// TIA Portal V16 program export: 3 tag tables, 3 data types, 3 data blocks, 6 code blocks (in call order from the OBs), 9 instance data blocks

VAR_GLOBAL   // PLC tag table "Entradas PLC"
   "Rele Emergencia" AT %I0.0 : Bool;
   "Rele Barrera" AT %I0.1 : Bool;
   "Pulsador Rearme" AT %I0.2 : Bool;
   "Marcha 1" AT %I0.3 : Bool;
   "Marcha 2" AT %I0.4 : Bool;
   "Marcha 3" AT %I0.5 : Bool;
   Caudalímetro AT %I0.6 : Bool;
   Presostato AT %I0.7 : Bool;
   "Final Soldadura" AT %I1.1 : Bool;
   "Soldadura RDY" AT %I1.0 : Bool;
   "Acuse error soldadura" AT %I1.2 : Bool;
   "Fibra óptica Tornillo 1" AT %I1.3 : Bool;
   "Fibra óptica Tornillo 2" AT %I1.4 : Bool;
   "Cajón rechazo" AT %I1.5 : Bool;
   "Pinza 1 RE" AT %I2.0 : Bool;
   "Pinza 1 AV" AT %I2.1 : Bool;
   "Pinza 2 RE" AT %I2.2 : Bool;
   "Pinza 2 AV" AT %I2.3 : Bool;
   "Pinza 3 RE" AT %I2.4 : Bool;
   "Pinza 3 AV" AT %I2.5 : Bool;
   "Libre I 2.6" AT %I2.6 : Bool;
   "Libre I 2.7" AT %I2.7 : Bool;
   "Selector acuse pieza mala" AT %I3.0 : Bool;
   RobotOK AT %I3.1 : Bool;
   RobotNOK AT %I3.2 : Bool;
   RobotAuto AT %I3.3 : Bool;
   "Libre I 3.4" AT %I3.4 : Bool;
   "Libre I 3.5" AT %I3.5 : Bool;
   "Libre I 3.6" AT %I3.6 : Bool;
   "Libre I 3.7" AT %I3.7 : Bool;
   Tag_71 AT %IW64 : Word;
END_VAR

VAR_GLOBAL   // PLC tag table "Salidas PLC"
   Rearme AT %Q0.0 : Bool;
   "Marcha Soldadura" AT %Q0.1 : Bool;
   "Programa 1" AT %Q0.2 : Bool;
   "Programa 2" AT %Q0.3 : Bool;
   "Programa 4" AT %Q0.4 : Bool;
   "Programa 8" AT %Q0.5 : Bool;
   "Programa 16" AT %Q0.6 : Bool;
   "Reset error" AT %Q0.7 : Bool;
   Fluorescent AT %Q1.0 : Bool;
   "Piloto 1 Rojo" AT %Q2.0 : Bool;
   "Piloto 1 Ambar" AT %Q2.1 : Bool;
   "Piloto 1 Verde" AT %Q2.2 : Bool;
   "Piloto 2 Rojo" AT %Q2.3 : Bool;
   "Piloto 2 Ambar" AT %Q2.4 : Bool;
   "Piloto 2 Verde" AT %Q2.5 : Bool;
   "Piloto 3 Rojo" AT %Q2.6 : Bool;
   "Piloto 3 Ambar" AT %Q2.7 : Bool;
   "Piloto 3 Verde" AT %Q3.0 : Bool;
   "Baliza Roja" AT %Q3.1 : Bool;
   "Baliza Ambar" AT %Q3.2 : Bool;
   "Baliza Verde" AT %Q3.3 : Bool;
   "Pinza 1" AT %Q4.0 : Bool;
   "Pinza 2" AT %Q4.1 : Bool;
   "Pinza 3" AT %Q4.2 : Bool;
   "Piloto Marcha 1" AT %Q3.5 : Bool;
   "Piloto Marcha 2" AT %Q3.6 : Bool;
   "Piloto Marcha 3" AT %Q3.7 : Bool;
   "Piloto rearme" AT %Q3.4 : Bool;
   "Libre Q 4.7" AT %Q4.7 : Bool;
   Tag_46 AT %Q1.1 : Bool;
   bNotReady AT %Q4.4 : Bool;
   bRobotReset AT %Q4.5 : Bool;
END_VAR

VAR_GLOBAL   // PLC tag table "Tabla de variables estándar"
   System_Byte AT %MB1001 : Byte;
   FirstScan AT %M1001.0 : Bool;
   DiagStatusUpdate AT %M1001.1 : Bool;
   AlwaysTRUE AT %M1001.2 : Bool;
   AlwaysFALSE AT %M1001.3 : Bool;
   Clock_Byte AT %MB1000 : Byte;
   Clock_10Hz AT %M1000.0 : Bool;
   Clock_5Hz AT %M1000.1 : Bool;
   "Clock_2.5Hz" AT %M1000.2 : Bool;
   Clock_2Hz AT %M1000.3 : Bool;
   "Clock_1.25Hz" AT %M1000.4 : Bool;
   Clock_1Hz AT %M1000.5 : Bool;
   "Clock_0.625Hz" AT %M1000.6 : Bool;
   "Clock_0.5Hz" AT %M1000.7 : Bool;
   Tag_1 AT %MW100 : Word;
   Tag_2 AT %M10.0 : Bool;
   bStartShortBolt AT %M20.0 : Bool;
   bStartMediumBolt AT %M20.1 : Bool;
   bStartLongBolt AT %M20.2 : Bool;
   bStartWeldingGripper_3 AT %M20.3 : Bool;
   bRetractGripper_3 AT %M20.4 : Bool;
   Tag_8 AT %M20.5 : Bool;
   Tag_9 AT %M20.6 : Bool;
   Tag_10 AT %M20.7 : Bool;
   bGripper_3_Conditions AT %M29.0 : Bool;
   bStartSmallNut AT %M21.0 : Bool;
   bStartBigNut AT %M21.1 : Bool;
   bStartWeldingGripper_2 AT %M21.2 : Bool;
   bRetractGripper_2 AT %M21.3 : Bool;
   Tag_16 AT %M21.4 : Bool;
   Tag_17 AT %M21.5 : Bool;
   Tag_18 AT %M21.6 : Bool;
   Tag_19 AT %M21.7 : Bool;
   bGripper_2_Conditions AT %M29.1 : Bool;
   bStartSpot AT %M22.0 : Bool;
   bStartWeldingGripper_1 AT %M22.1 : Bool;
   bRetractGripper_1 AT %M22.2 : Bool;
   Tag_24 AT %M22.3 : Bool;
   Tag_25 AT %M22.4 : Bool;
   Tag_26 AT %M22.5 : Bool;
   Tag_27 AT %M22.6 : Bool;
   Tag_28 AT %M22.7 : Bool;
   bGripper_1_Conditions AT %M29.2 : Bool;
   bCycleConditions AT %M29.3 : Bool;
   bEndOfCycle AT %M23.0 : Bool;
   bWeldingNOK AT %M23.1 : Bool;
   bToScrap AT %M23.2 : Bool;
   bScraped AT %M23.3 : Bool;
   bScrapBoxFull AT %M23.4 : Bool;
   bConsecutiveNOKtoBlock AT %M23.5 : Bool;
   bRobotAuto AT %M23.6 : Bool;
   bProductionCompleted AT %M23.7 : Bool;
   bAction_1 AT %M24.0 : Bool;
   bAction_2 AT %M24.1 : Bool;
   bAction_3 AT %M24.2 : Bool;
   bAction_4 AT %M24.3 : Bool;
   bAction_5 AT %M24.4 : Bool;
   bAction_6 AT %M24.5 : Bool;
   bEndSequence AT %M24.6 : Bool;
   BWelderProgNumber AT %MB12 : Byte;
   bWelderProg_Bit_0 AT %M12.0 : Bool;
   bWelderProg_Bit_1 AT %M12.1 : Bool;
   bWelderProg_Bit_2 AT %M12.2 : Bool;
   bWelderProg_Bit_3 AT %M12.3 : Bool;
   bWelderProg_Bit_4 AT %M12.4 : Bool;
   Tag_53 AT %MW20 : Int;
   Tag_54 AT %MW22 : Int;
   Tag_55 AT %MW24 : Int;
   "Alarmes 1" AT %MW200 : Word;
   "Alarmes 2" AT %MW202 : Word;
   bAnyAlarm AT %M210.0 : Bool;
   Tag_59 AT %MD200 : DWord;
   bEmergenciesNOK AT %M200.0 : Bool;
   bPressureFault AT %M200.1 : Bool;
   bFlowFault AT %M200.2 : Bool;
   "Alarma barrera cajon rechazo" AT %M200.3 : Bool;
   "Alarma pinza 1 no avanza" AT %M201.0 : Bool;
   "Alarma pinza 1 No retrocede" AT %M201.1 : Bool;
   "Alarma pinza 2 No avanza" AT %M201.2 : Bool;
   "Alarma pinza 2 No retrocede" AT %M201.3 : Bool;
   "Alarma pinza3 no avanza" AT %M201.4 : Bool;
   "Alarma pinza 3 No retrocede" AT %M201.5 : Bool;
   bWelderNotReady AT %M200.4 : Bool;
   bWelderNotResponding AT %M200.5 : Bool;
   "Alarma barrera obstruida" AT %M202.0 : Bool;
   Tag_73 AT %M200.6 : Bool;
   "Aviso perno corto incorreto" AT %M202.1 : Bool;
   "Aviso perno medio incorrecto" AT %M202.2 : Bool;
   "Aviso perno largo incorrecto" AT %M202.3 : Bool;
   "Aviso pieza mala" AT %M202.4 : Bool;
   "Aviso tirar pieza mala" AT %M202.5 : Bool;
   Tag_79 AT %M202.6 : Bool;
   bInitConditions AT %M29.4 : Bool;
   "Alarmes 6" AT %MW210 : Word;
   Tag_56 AT %M200.7 : Bool;
   Tag_57 AT %M5.0 : Bool;
   Tag_60 AT %M5.1 : Bool;
   Tag_61 AT %M5.2 : Bool;
   Tag_62 AT %M5.3 : Bool;
   Tag_63 AT %M5.4 : Bool;
   Tag_64 AT %M5.5 : Bool;
   Tag_58 AT %M7.0 : Bool;
   Tag_65 AT %M6.5 : Bool;
   Tag_66 AT %M6.4 : Bool;
   Tag_67 AT %M6.2 : Bool;
   Tag_68 AT %M6.3 : Bool;
   Tag_69 AT %M6.0 : Bool;
   Tag_70 AT %M6.1 : Bool;
   bTemp_PAP AT %M100.0 : Bool;
   bRedLamp_3_NonInverted AT %M50.0 : Bool;
   bRedLamp_1_Inverted AT %M50.1 : Bool;
   bAmberLamp_3_NonInverted AT %M50.2 : Bool;
   bGreenLamp_3_NonInverted AT %M50.4 : Bool;
   bAmberLamp_1_Inverted AT %M50.3 : Bool;
   bGreenLamp_1_Inverted AT %M50.5 : Bool;
   bRedLamp_1_NonInverted AT %M50.6 : Bool;
   bRedLamp_3_Inverted AT %M50.7 : Bool;
   bAmberLamp_1_NonInverted AT %M51.0 : Bool;
   bAmberLamp_3_Inverted AT %M51.1 : Bool;
   bGreenLamp_1_NonInverted AT %M51.2 : Bool;
   bGreenLamp_3_Inverted AT %M51.3 : Bool;
   bStartLamp_1_NonInverted AT %M51.4 : Bool;
   bStartLamp_3_NonInverted AT %M51.5 : Bool;
   bStartLamp_3_Inverted AT %M51.6 : Bool;
   bStartLamp_1_Inverted AT %M51.7 : Bool;
   bGripper_3_NonInverted AT %M52.0 : Bool;
   bGripper_1_NonInverted AT %M52.1 : Bool;
   bGripper_3_Inverted AT %M52.3 : Bool;
   bGripper_1_Inverted AT %M52.2 : Bool;
END_VAR

TYPE "udtCounters"
// stored: IsFailsafeCompliant false
   STRUCT
      diPreselectionValue : DInt;
      diTotalOK : DInt;
      diPartialOK : DInt;
      diConsecutiveOK : DInt;
      diTotalNOK : DInt;
      diPartialNOK : DInt;
      diConsecutiveNOK : DInt;
      diScrapBox : DInt;
      stSettings : Struct
         diScrapBoxSize : DInt;
         diNOKValueToBlock : DInt;
         diOKValueToResetNOK : DInt;
      END_STRUCT;
      stButtons : Struct
         bResetTotalOK : Bool;
         bResetPartialOK : Bool;
         bResetConsecutiveOK : Bool;
         bResetTotalNOK : Bool;
         bResetPartialNOK : Bool;
         bResetConsecutiveNOK : Bool;
         bResetScrapBox : Bool;
      END_STRUCT;
   END_STRUCT;
END_TYPE

TYPE "udtProgram"
// stored: IsFailsafeCompliant false
   STRUCT
      strName : String[12];
      udtStep { S7_SetPoint := 'True'} : Array[1..10] of "udtStep";
      udtCounter { S7_SetPoint := 'True'} : "udtCounters";
   END_STRUCT;
END_TYPE

TYPE "udtStep"
// stored: IsFailsafeCompliant false
   STRUCT
      iAction : Int;
      iPG : Int;
      iLamp : Int;
   END_STRUCT;
END_TYPE

DATA_BLOCK "db_HMI"   // DB100
{ S7_Optimized_Access := 'FALSE' }
VERSION : 0.1
// stored: AutoNumber false, IsOnlyStoredInLoadMemory false, IsWriteProtectedInAS false
   VAR
      ariScreen : Array[0..3] of Int;
      iScreenNumbver : Int;
      bLights : Bool;
      bResetCycleKey : Bool;
      diPartsCounter : DInt;
      iPart_1 : Int;
      iPart_2 : Int;
      iPart_3 : Int;
      iPart_4 : Int;
      iPart_5 : Int;
      iPart_6 : Int;
      iPart_7 : Int;
      iPart_8 : Int;
      iPart_9 : Int;
      iPart_10 : Int;
   END_VAR
BEGIN
END_DATA_BLOCK

DATA_BLOCK "db_Programs"   // DB101
{ S7_Optimized_Access := 'TRUE' }
VERSION : 0.1
// stored: AutoNumber false, IsOnlyStoredInLoadMemory false, IsRetainMemResEnabled false, IsWriteProtectedInAS false, MemoryReserve 100
   VAR RETAIN
      diProgramSelection : DInt := 8;
   END_VAR
   VAR
      bSaveKey : Bool := FALSE;
      diStepCounter : DInt := 1;
      strShortBolt : String[16] := '';
      strMediumBolt : String[16] := '';
      strLongBolt : String[16] := '';
      strSmallNut : String[16] := '';
      strBigNut : String[16] := '';
   END_VAR
   VAR RETAIN
      udtProgram { S7_SetPoint := 'True'} : Array[1..10] of "udtProgram";
      udtWorkProgram { S7_SetPoint := 'True'} : "udtProgram";
   END_VAR
   VAR
      udtWorkStep { S7_SetPoint := 'True'} : "udtStep";
   END_VAR
BEGIN
   udtProgram[1].strName := 'TCS327=178';
   udtProgram[2].strName := 'TCS327=193';
   udtProgram[3].strName := 'TCS327=192';
   udtProgram[4].strName := 'TCS327=181';
   udtProgram[5].strName := 'TCS327=186';
   udtProgram[6].strName := 'TCS327=200';
   udtProgram[7].strName := 'TCS327=188';
   udtProgram[8].strName := 'TCS327=190';
   udtProgram[9].strName := 'TCS327=197';
   udtProgram[10].strName := '191.33476980';
   udtProgram[1].udtStep[1..4].iAction := 2;
   udtProgram[1].udtStep[5..7].iAction := 1;
   udtProgram[1].udtStep[8..10].iAction := 0;
   udtProgram[2].udtStep[1].iAction := 6;
   udtProgram[2].udtStep[2].iAction := 5;
   udtProgram[2].udtStep[3..4].iAction := 3;
   udtProgram[2].udtStep[5..10].iAction := 0;
   udtProgram[3].udtStep[1..2].iAction := 1;
   udtProgram[3].udtStep[3..10].iAction := 0;
   udtProgram[4].udtStep[1..3].iAction := 6;
   udtProgram[4].udtStep[4].iAction := 1;
   udtProgram[4].udtStep[5..10].iAction := 0;
   udtProgram[5].udtStep[1..2].iAction := 2;
   udtProgram[5].udtStep[3..10].iAction := 0;
   udtProgram[6].udtStep[1].iAction := 5;
   udtProgram[6].udtStep[2].iAction := 1;
   udtProgram[6].udtStep[3..10].iAction := 0;
   udtProgram[7].udtStep[1].iAction := 5;
   udtProgram[7].udtStep[2].iAction := 1;
   udtProgram[7].udtStep[3..10].iAction := 0;
   udtProgram[8].udtStep[1].iAction := 6;
   udtProgram[8].udtStep[2].iAction := 4;
   udtProgram[8].udtStep[3..7].iAction := 1;
   udtProgram[8].udtStep[8..10].iAction := 0;
   udtProgram[9].udtStep[1..3].iAction := 4;
   udtProgram[9].udtStep[4..10].iAction := 0;
   udtProgram[10].udtStep[1..10].iAction := 0;
   udtProgram[1].udtStep[1..7].iPG := 3;
   udtProgram[1].udtStep[8..10].iPG := 0;
   udtProgram[2].udtStep[1].iPG := 22;
   udtProgram[2].udtStep[2].iPG := 23;
   udtProgram[2].udtStep[3..4].iPG := 3;
   udtProgram[2].udtStep[5].iPG := 9;
   udtProgram[2].udtStep[6..7].iPG := 1;
   udtProgram[2].udtStep[8..10].iPG := 0;
   udtProgram[3].udtStep[1..2].iPG := 3;
   udtProgram[3].udtStep[3..10].iPG := 0;
   udtProgram[4].udtStep[1..3].iPG := 22;
   udtProgram[4].udtStep[4].iPG := 3;
   udtProgram[4].udtStep[5..10].iPG := 0;
   udtProgram[5].udtStep[1..3].iPG := 3;
   udtProgram[5].udtStep[4..10].iPG := 0;
   udtProgram[6].udtStep[1].iPG := 5;
   udtProgram[6].udtStep[2].iPG := 3;
   udtProgram[6].udtStep[3..10].iPG := 0;
   udtProgram[7].udtStep[1].iPG := 5;
   udtProgram[7].udtStep[2].iPG := 3;
   udtProgram[7].udtStep[3..10].iPG := 0;
   udtProgram[8].udtStep[1].iPG := 1;
   udtProgram[8].udtStep[2].iPG := 2;
   udtProgram[8].udtStep[3..7].iPG := 3;
   udtProgram[8].udtStep[8..10].iPG := 0;
   udtProgram[9].udtStep[1..3].iPG := 1;
   udtProgram[9].udtStep[4..10].iPG := 0;
   udtProgram[10].udtStep[1..10].iPG := 0;
   udtProgram[1].udtStep[1].iLamp := 2;
   udtProgram[1].udtStep[2].iLamp := 1;
   udtProgram[1].udtStep[3].iLamp := 3;
   udtProgram[1].udtStep[4].iLamp := 4;
   udtProgram[1].udtStep[5].iLamp := 5;
   udtProgram[1].udtStep[6].iLamp := 6;
   udtProgram[1].udtStep[7].iLamp := 7;
   udtProgram[1].udtStep[8..10].iLamp := 0;
   udtProgram[2].udtStep[1..2].iLamp := 2;
   udtProgram[2].udtStep[3].iLamp := 3;
   udtProgram[2].udtStep[4].iLamp := 4;
   udtProgram[2].udtStep[5].iLamp := 5;
   udtProgram[2].udtStep[6].iLamp := 6;
   udtProgram[2].udtStep[7].iLamp := 7;
   udtProgram[2].udtStep[8..10].iLamp := 0;
   udtProgram[3].udtStep[1].iLamp := 1;
   udtProgram[3].udtStep[2].iLamp := 2;
   udtProgram[3].udtStep[3..10].iLamp := 0;
   udtProgram[4].udtStep[1].iLamp := 1;
   udtProgram[4].udtStep[2].iLamp := 2;
   udtProgram[4].udtStep[3].iLamp := 3;
   udtProgram[4].udtStep[4..10].iLamp := 0;
   udtProgram[5].udtStep[1].iLamp := 1;
   udtProgram[5].udtStep[2].iLamp := 2;
   udtProgram[5].udtStep[3].iLamp := 3;
   udtProgram[5].udtStep[4..10].iLamp := 0;
   udtProgram[6].udtStep[1].iLamp := 1;
   udtProgram[6].udtStep[2].iLamp := 2;
   udtProgram[6].udtStep[3..10].iLamp := 0;
   udtProgram[7].udtStep[1].iLamp := 1;
   udtProgram[7].udtStep[2].iLamp := 2;
   udtProgram[7].udtStep[3..10].iLamp := 0;
   udtProgram[8].udtStep[1].iLamp := 7;
   udtProgram[8].udtStep[2].iLamp := 1;
   udtProgram[8].udtStep[3].iLamp := 6;
   udtProgram[8].udtStep[4].iLamp := 5;
   udtProgram[8].udtStep[5].iLamp := 3;
   udtProgram[8].udtStep[6].iLamp := 2;
   udtProgram[8].udtStep[7].iLamp := 4;
   udtProgram[8].udtStep[8..10].iLamp := 0;
   udtProgram[9].udtStep[1].iLamp := 1;
   udtProgram[9].udtStep[2].iLamp := 2;
   udtProgram[9].udtStep[3].iLamp := 3;
   udtProgram[9].udtStep[4..10].iLamp := 0;
   udtProgram[10].udtStep[1..10].iLamp := 0;
   udtWorkProgram.strName := 'TCS327=190';
   udtWorkProgram.udtStep[1].iAction := 6;
   udtWorkProgram.udtStep[2].iAction := 4;
   udtWorkProgram.udtStep[3..7].iAction := 1;
   udtWorkProgram.udtStep[8..10].iAction := 0;
   udtWorkProgram.udtStep[1].iPG := 1;
   udtWorkProgram.udtStep[2].iPG := 2;
   udtWorkProgram.udtStep[3..7].iPG := 3;
   udtWorkProgram.udtStep[8..10].iPG := 0;
   udtWorkProgram.udtStep[1].iLamp := 7;
   udtWorkProgram.udtStep[2].iLamp := 1;
   udtWorkProgram.udtStep[3].iLamp := 6;
   udtWorkProgram.udtStep[4].iLamp := 5;
   udtWorkProgram.udtStep[5].iLamp := 3;
   udtWorkProgram.udtStep[6].iLamp := 2;
   udtWorkProgram.udtStep[7].iLamp := 4;
   udtWorkProgram.udtStep[8..10].iLamp := 0;
   udtWorkStep.iAction := 6;
   udtWorkStep.iPG := 1;
   udtWorkStep.iLamp := 7;
END_DATA_BLOCK

DATA_BLOCK "db_Settings"   // DB2
{ S7_Optimized_Access := 'TRUE' }
VERSION : 0.1
// stored: AutoNumber true, IsOnlyStoredInLoadMemory false, IsRetainMemResEnabled false, IsWriteProtectedInAS false, MemoryReserve 100
   VAR RETAIN
      bIsInverted : Bool;
   END_VAR
   VAR
      bBypasRobot : Bool;
   END_VAR
   VAR RETAIN
      iSerialNumber : Int;
   END_VAR
BEGIN
END_DATA_BLOCK

ORGANIZATION_BLOCK "Main"   // OB1, LAD, ProgramCycle
TITLE = "Main Program Sweep (Cycle)"
{ S7_Optimized_Access := 'TRUE' }
VERSION : 0.1
// stored: AutoNumber true, IsIECCheckEnabled false, SetENOAutomatically false
   VAR_INPUT
      Initial_Call : Bool;   // Initial call of this OB
      Remanence : Bool;   // =True, if remanent data are available
   END_VAR
BEGIN

REGION Network 1
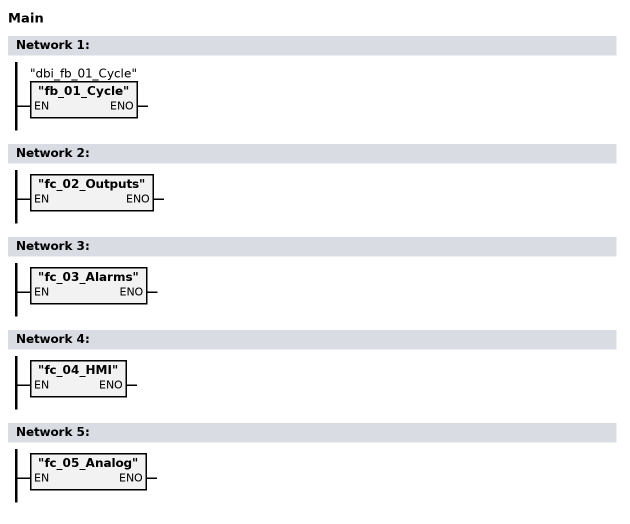
   RUNG wire#powerrail
      "dbi_fb_01_Cycle"()
   END_RUNG
   // the same network as SCL:
   "dbi_fb_01_Cycle"();   // "fb_01_Cycle"
END_REGION

REGION Network 2
   RUNG wire#powerrail
      "fc_02_Outputs"()
   END_RUNG
   // the same network as SCL:
   "fc_02_Outputs"();
END_REGION

REGION Network 3
   RUNG wire#powerrail
      "fc_03_Alarms"()
   END_RUNG
   // the same network as SCL:
   "fc_03_Alarms"();
END_REGION

REGION Network 4
   RUNG wire#powerrail
      "fc_04_HMI"()
   END_RUNG
   // the same network as SCL:
   "fc_04_HMI"();
END_REGION

REGION Network 5
   RUNG wire#powerrail
      "fc_05_Analog"()
   END_RUNG
   // the same network as SCL:
   "fc_05_Analog"();
END_REGION
END_ORGANIZATION_BLOCK

FUNCTION_BLOCK "fb_01_Cycle"   // FB1, LAD
{ S7_Optimized_Access := 'TRUE' }
VERSION : 0.1
// stored: AutoNumber false, IsIECCheckEnabled false, IsRetainMemResEnabled false, MemoryReserve 100, SetENOAutomatically false, UDAEnableTagReadback false
   VAR
      TON_Delay : Array[1..10] of TON_TIME;
      TP_Reset { S7_SetPoint := 'True'} : TP_TIME;
   END_VAR
   VAR_TEMP
      bBypassRobot : Bool;
      bRobotReset : Bool;
      bIsInverted : Bool;
   END_VAR
   VAR_TEMP   // added for the SCL form of the ladder/FBD networks
      _w1 : Bool;
      _w2 : Bool;
   END_VAR
BEGIN

REGION Network 1: Reseteo Ciclos por Emergencias
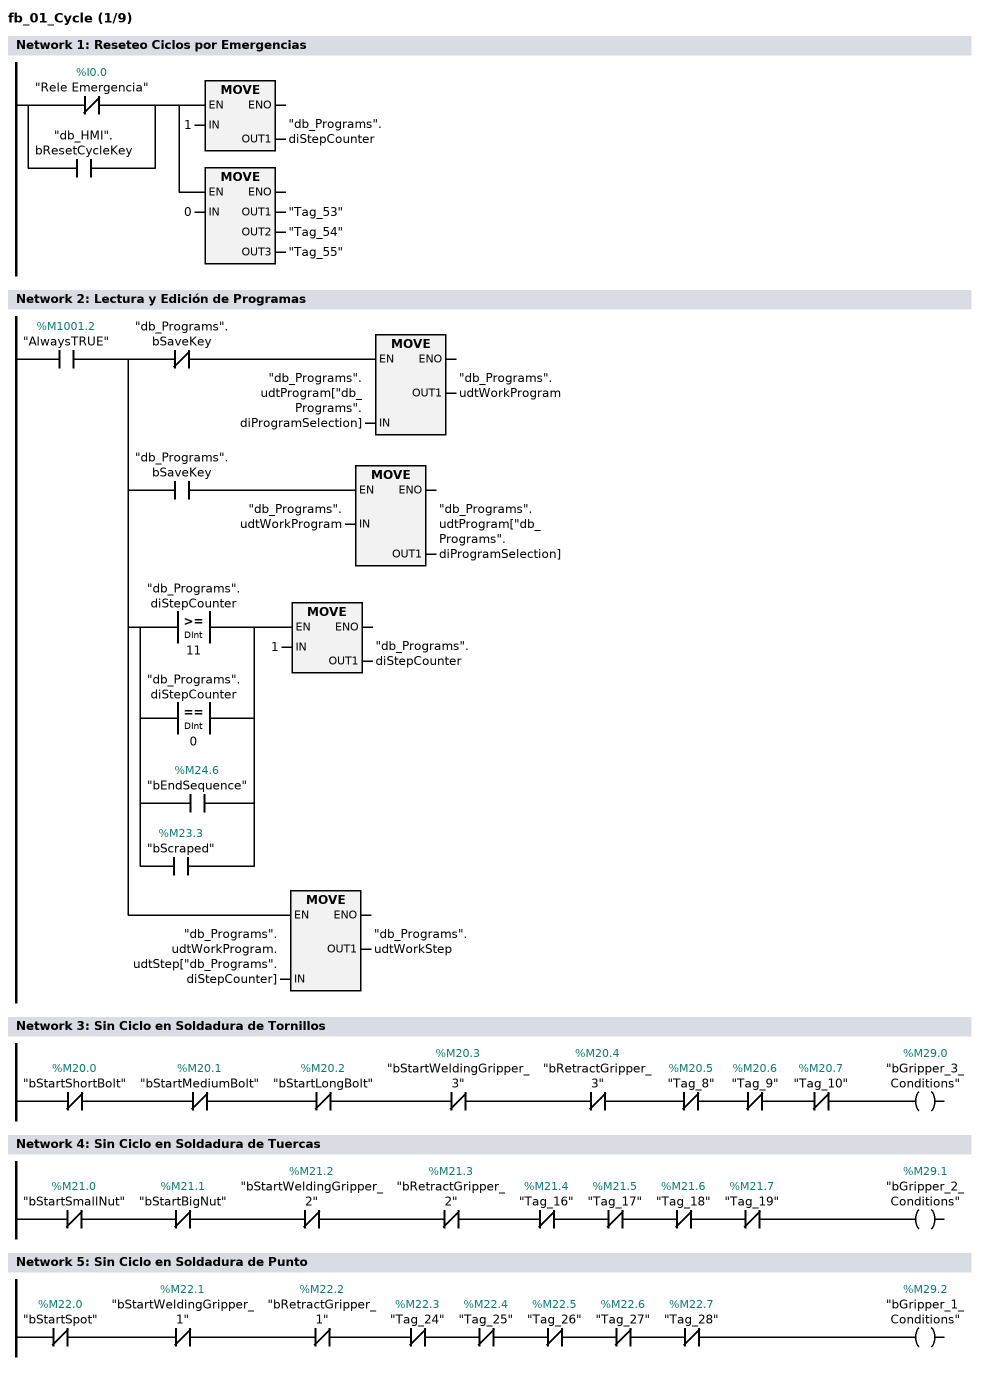
   RUNG wire#powerrail
      I_Contact( "Rele Emergencia" )
      wire#w1
      Move(in := 1, out1 => "db_Programs".diStepCounter)
   END_RUNG
   RUNG wire#powerrail
      Contact( "db_HMI".bResetCycleKey )
   END_RUNG wire#w1
   RUNG wire#w1
      Move(in := 0, out1 => "Tag_53", out2 => "Tag_54", out3 => "Tag_55")
   END_RUNG
   // the same network as SCL:
   IF NOT "Rele Emergencia" OR "db_HMI".bResetCycleKey THEN
       "db_Programs".diStepCounter := 1;
       "Tag_53" := 0;
       "Tag_54" := 0;
       "Tag_55" := 0;
   END_IF;
END_REGION

REGION Network 2: Lectura y Edición de Programas
   RUNG wire#powerrail
      Contact( "AlwaysTRUE" )
      wire#w1
      I_Contact( "db_Programs".bSaveKey )
      Move(in := "db_Programs".udtProgram["db_Programs".diProgramSelection], out1 => "db_Programs".udtWorkProgram)
   END_RUNG
   RUNG wire#w1
      Contact( "db_Programs".bSaveKey )
      Move(in := "db_Programs".udtWorkProgram, out1 => "db_Programs".udtProgram["db_Programs".diProgramSelection])
   END_RUNG
   RUNG wire#w1
      { S7_Templates := "SrcType := DInt" } GE_Contact(in1 := "db_Programs".diStepCounter, in2 := 11)
      wire#w2
      Move(in := 1, out1 => "db_Programs".diStepCounter)
   END_RUNG
   RUNG wire#w1
      { S7_Templates := "SrcType := DInt" } EQ_Contact(in1 := "db_Programs".diStepCounter, in2 := 0)
   END_RUNG wire#w2
   RUNG wire#w1
      Contact( "bEndSequence" )
   END_RUNG wire#w2
   RUNG wire#w1
      Contact( "bScraped" )
   END_RUNG wire#w2
   RUNG wire#w1
      Move(in := "db_Programs".udtWorkProgram.udtStep["db_Programs".diStepCounter], out1 => "db_Programs".udtWorkStep)
   END_RUNG
   // the same network as SCL:
   IF "AlwaysTRUE" AND NOT "db_Programs".bSaveKey THEN
       "db_Programs".udtWorkProgram := "db_Programs".udtProgram["db_Programs".diProgramSelection];
   END_IF;
   IF "AlwaysTRUE" AND "db_Programs".bSaveKey THEN
       "db_Programs".udtProgram["db_Programs".diProgramSelection] := "db_Programs".udtWorkProgram;
   END_IF;
   IF "AlwaysTRUE" AND (("db_Programs".diStepCounter >= 11) OR ("db_Programs".diStepCounter = 0) OR "bEndSequence" OR "bScraped") THEN
       "db_Programs".diStepCounter := 1;
   END_IF;
   IF "AlwaysTRUE" THEN
       "db_Programs".udtWorkStep := "db_Programs".udtWorkProgram.udtStep["db_Programs".diStepCounter];
   END_IF;
END_REGION

REGION Network 3: Sin Ciclo en Soldadura de Tornillos
   RUNG wire#powerrail
      I_Contact( "bStartShortBolt" )
      I_Contact( "bStartMediumBolt" )
      I_Contact( "bStartLongBolt" )
      I_Contact( "bStartWeldingGripper_3" )
      I_Contact( "bRetractGripper_3" )
      I_Contact( "Tag_8" )
      I_Contact( "Tag_9" )
      I_Contact( "Tag_10" )
      Coil( "bGripper_3_Conditions" )
   END_RUNG
   // the same network as SCL:
   "bGripper_3_Conditions" := NOT "bStartShortBolt" AND NOT "bStartMediumBolt" AND NOT "bStartLongBolt" AND NOT "bStartWeldingGripper_3" AND NOT "bRetractGripper_3" AND NOT "Tag_8" AND NOT "Tag_9" AND NOT "Tag_10";
END_REGION

REGION Network 4: Sin Ciclo en Soldadura de Tuercas
   RUNG wire#powerrail
      I_Contact( "bStartSmallNut" )
      I_Contact( "bStartBigNut" )
      I_Contact( "bStartWeldingGripper_2" )
      I_Contact( "bRetractGripper_2" )
      I_Contact( "Tag_16" )
      I_Contact( "Tag_17" )
      I_Contact( "Tag_18" )
      I_Contact( "Tag_19" )
      Coil( "bGripper_2_Conditions" )
   END_RUNG
   // the same network as SCL:
   "bGripper_2_Conditions" := NOT "bStartSmallNut" AND NOT "bStartBigNut" AND NOT "bStartWeldingGripper_2" AND NOT "bRetractGripper_2" AND NOT "Tag_16" AND NOT "Tag_17" AND NOT "Tag_18" AND NOT "Tag_19";
END_REGION

REGION Network 5: Sin Ciclo en Soldadura de Punto
   RUNG wire#powerrail
      I_Contact( "bStartSpot" )
      I_Contact( "bStartWeldingGripper_1" )
      I_Contact( "bRetractGripper_1" )
      I_Contact( "Tag_24" )
      I_Contact( "Tag_25" )
      I_Contact( "Tag_26" )
      I_Contact( "Tag_27" )
      I_Contact( "Tag_28" )
      Coil( "bGripper_1_Conditions" )
   END_RUNG
   // the same network as SCL:
   "bGripper_1_Conditions" := NOT "bStartSpot" AND NOT "bStartWeldingGripper_1" AND NOT "bRetractGripper_1" AND NOT "Tag_24" AND NOT "Tag_25" AND NOT "Tag_26" AND NOT "Tag_27" AND NOT "Tag_28";
END_REGION

REGION Network 6: Condiciones Ciclo Auxiliares
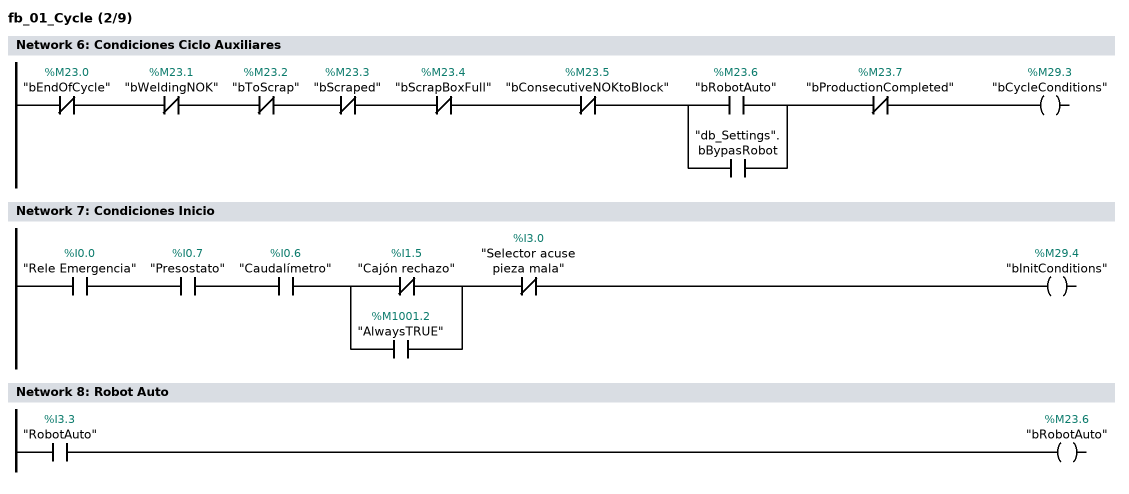
   RUNG wire#powerrail
      I_Contact( "bEndOfCycle" )
      I_Contact( "bWeldingNOK" )
      I_Contact( "bToScrap" )
      I_Contact( "bScraped" )
      I_Contact( "bScrapBoxFull" )
      I_Contact( "bConsecutiveNOKtoBlock" )
      wire#w1
      Contact( "bRobotAuto" )
      wire#w2
      I_Contact( "bProductionCompleted" )
      Coil( "bCycleConditions" )
   END_RUNG
   RUNG wire#w1
      Contact( "db_Settings".bBypasRobot )
   END_RUNG wire#w2
   // the same network as SCL:
   "bCycleConditions" := NOT "bEndOfCycle" AND NOT "bWeldingNOK" AND NOT "bToScrap" AND NOT "bScraped" AND NOT "bScrapBoxFull" AND NOT "bConsecutiveNOKtoBlock" AND ("bRobotAuto" OR "db_Settings".bBypasRobot) AND NOT "bProductionCompleted";
END_REGION

REGION Network 7: Condiciones Inicio
   RUNG wire#powerrail
      Contact( "Rele Emergencia" )
      Contact( "Presostato" )
      Contact( "Caudalímetro" )
      wire#w1
      I_Contact( "Cajón rechazo" )
      wire#w2
      I_Contact( "Selector acuse pieza mala" )
      Coil( "bInitConditions" )
   END_RUNG
   RUNG wire#w1
      Contact( "AlwaysTRUE" )
   END_RUNG wire#w2
   // the same network as SCL:
   "bInitConditions" := "Rele Emergencia" AND "Presostato" AND "Caudalímetro" AND (NOT "Cajón rechazo" OR "AlwaysTRUE") AND NOT "Selector acuse pieza mala";
END_REGION

REGION Network 8: Robot Auto
   RUNG wire#powerrail
      Contact( "RobotAuto" )
      Coil( "bRobotAuto" )
   END_RUNG
   // the same network as SCL:
   "bRobotAuto" := "RobotAuto";
END_REGION

REGION Network 9: Selección Acción
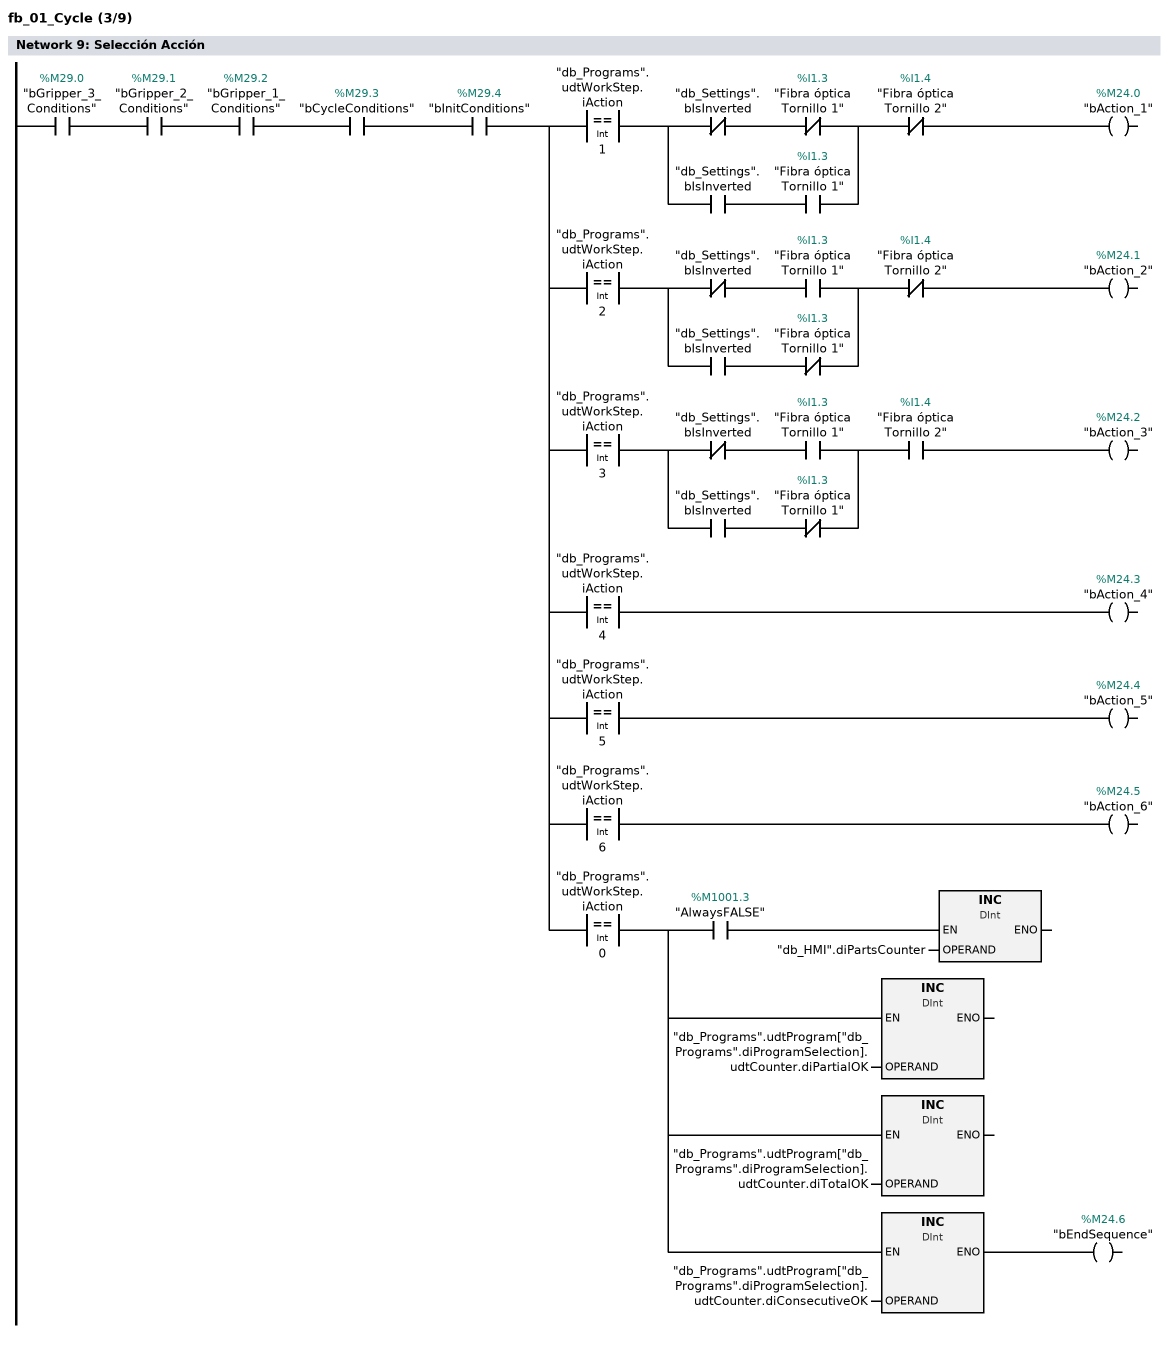
   RUNG wire#powerrail
      Contact( "bGripper_3_Conditions" )
      Contact( "bGripper_2_Conditions" )
      Contact( "bGripper_1_Conditions" )
      Contact( "bCycleConditions" )
      Contact( "bInitConditions" )
      wire#w1
      { S7_Templates := "SrcType := Int" } EQ_Contact(in1 := "db_Programs".udtWorkStep.iAction, in2 := 1)
      wire#w2
      I_Contact( "db_Settings".bIsInverted )
      I_Contact( "Fibra óptica Tornillo 1" )
      wire#w3
      I_Contact( "Fibra óptica Tornillo 2" )
      Coil( "bAction_1" )
   END_RUNG
   RUNG wire#w2
      Contact( "db_Settings".bIsInverted )
      Contact( "Fibra óptica Tornillo 1" )
   END_RUNG wire#w3
   RUNG wire#w1
      { S7_Templates := "SrcType := Int" } EQ_Contact(in1 := "db_Programs".udtWorkStep.iAction, in2 := 2)
      wire#w4
      I_Contact( "db_Settings".bIsInverted )
      Contact( "Fibra óptica Tornillo 1" )
      wire#w5
      I_Contact( "Fibra óptica Tornillo 2" )
      Coil( "bAction_2" )
   END_RUNG
   RUNG wire#w4
      Contact( "db_Settings".bIsInverted )
      I_Contact( "Fibra óptica Tornillo 1" )
   END_RUNG wire#w5
   RUNG wire#w1
      { S7_Templates := "SrcType := Int" } EQ_Contact(in1 := "db_Programs".udtWorkStep.iAction, in2 := 3)
      wire#w6
      I_Contact( "db_Settings".bIsInverted )
      Contact( "Fibra óptica Tornillo 1" )
      wire#w7
      Contact( "Fibra óptica Tornillo 2" )
      Coil( "bAction_3" )
   END_RUNG
   RUNG wire#w6
      Contact( "db_Settings".bIsInverted )
      I_Contact( "Fibra óptica Tornillo 1" )
   END_RUNG wire#w7
   RUNG wire#w1
      { S7_Templates := "SrcType := Int" } EQ_Contact(in1 := "db_Programs".udtWorkStep.iAction, in2 := 4)
      Coil( "bAction_4" )
   END_RUNG
   RUNG wire#w1
      { S7_Templates := "SrcType := Int" } EQ_Contact(in1 := "db_Programs".udtWorkStep.iAction, in2 := 5)
      Coil( "bAction_5" )
   END_RUNG
   RUNG wire#w1
      { S7_Templates := "SrcType := Int" } EQ_Contact(in1 := "db_Programs".udtWorkStep.iAction, in2 := 6)
      Coil( "bAction_6" )
   END_RUNG
   RUNG wire#w1
      { S7_Templates := "SrcType := Int" } EQ_Contact(in1 := "db_Programs".udtWorkStep.iAction, in2 := 0)
      wire#w8
      Contact( "AlwaysFALSE" )
      { S7_Templates := "DestType := DInt" } Inc( "db_HMI".diPartsCounter )
   END_RUNG
   RUNG wire#w8
      { S7_Templates := "DestType := DInt" } Inc( "db_Programs".udtProgram["db_Programs".diProgramSelection].udtCounter.diPartialOK )
   END_RUNG
   RUNG wire#w8
      { S7_Templates := "DestType := DInt" } Inc( "db_Programs".udtProgram["db_Programs".diProgramSelection].udtCounter.diTotalOK )
   END_RUNG
   RUNG wire#w8
      { S7_Templates := "DestType := DInt" } Inc( "db_Programs".udtProgram["db_Programs".diProgramSelection].udtCounter.diConsecutiveOK )
      Coil( "bEndSequence" )
   END_RUNG
   // the same network as SCL:
   #_w1 := "bGripper_3_Conditions" AND "bGripper_2_Conditions" AND "bGripper_1_Conditions" AND "bCycleConditions" AND "bInitConditions";
   "bAction_1" := #_w1 AND ("db_Programs".udtWorkStep.iAction = 1) AND ((NOT "db_Settings".bIsInverted AND NOT "Fibra óptica Tornillo 1") OR ("db_Settings".bIsInverted AND "Fibra óptica Tornillo 1")) AND NOT "Fibra óptica Tornillo 2";
   "bAction_2" := #_w1 AND ("db_Programs".udtWorkStep.iAction = 2) AND ((NOT "db_Settings".bIsInverted AND "Fibra óptica Tornillo 1") OR ("db_Settings".bIsInverted AND NOT "Fibra óptica Tornillo 1")) AND NOT "Fibra óptica Tornillo 2";
   "bAction_3" := #_w1 AND ("db_Programs".udtWorkStep.iAction = 3) AND ((NOT "db_Settings".bIsInverted AND "Fibra óptica Tornillo 1") OR ("db_Settings".bIsInverted AND NOT "Fibra óptica Tornillo 1")) AND "Fibra óptica Tornillo 2";
   "bAction_4" := #_w1 AND ("db_Programs".udtWorkStep.iAction = 4);
   "bAction_5" := #_w1 AND ("db_Programs".udtWorkStep.iAction = 5);
   "bAction_6" := #_w1 AND ("db_Programs".udtWorkStep.iAction = 6);
   #_w2 := #_w1 AND ("db_Programs".udtWorkStep.iAction = 0);
   IF #_w2 AND "AlwaysFALSE" THEN "db_HMI".diPartsCounter := "db_HMI".diPartsCounter + 1; END_IF;
   IF #_w2 THEN
       "db_Programs".udtProgram["db_Programs".diProgramSelection].udtCounter.diPartialOK := "db_Programs".udtProgram["db_Programs".diProgramSelection].udtCounter.diPartialOK + 1;
       "db_Programs".udtProgram["db_Programs".diProgramSelection].udtCounter.diTotalOK := "db_Programs".udtProgram["db_Programs".diProgramSelection].udtCounter.diTotalOK + 1;
       "db_Programs".udtProgram["db_Programs".diProgramSelection].udtCounter.diConsecutiveOK := "db_Programs".udtProgram["db_Programs".diProgramSelection].udtCounter.diConsecutiveOK + 1;
   END_IF;
   "bEndSequence" := #_w2;
END_REGION

REGION Network 10: Orden Inicio Tornillo Corto
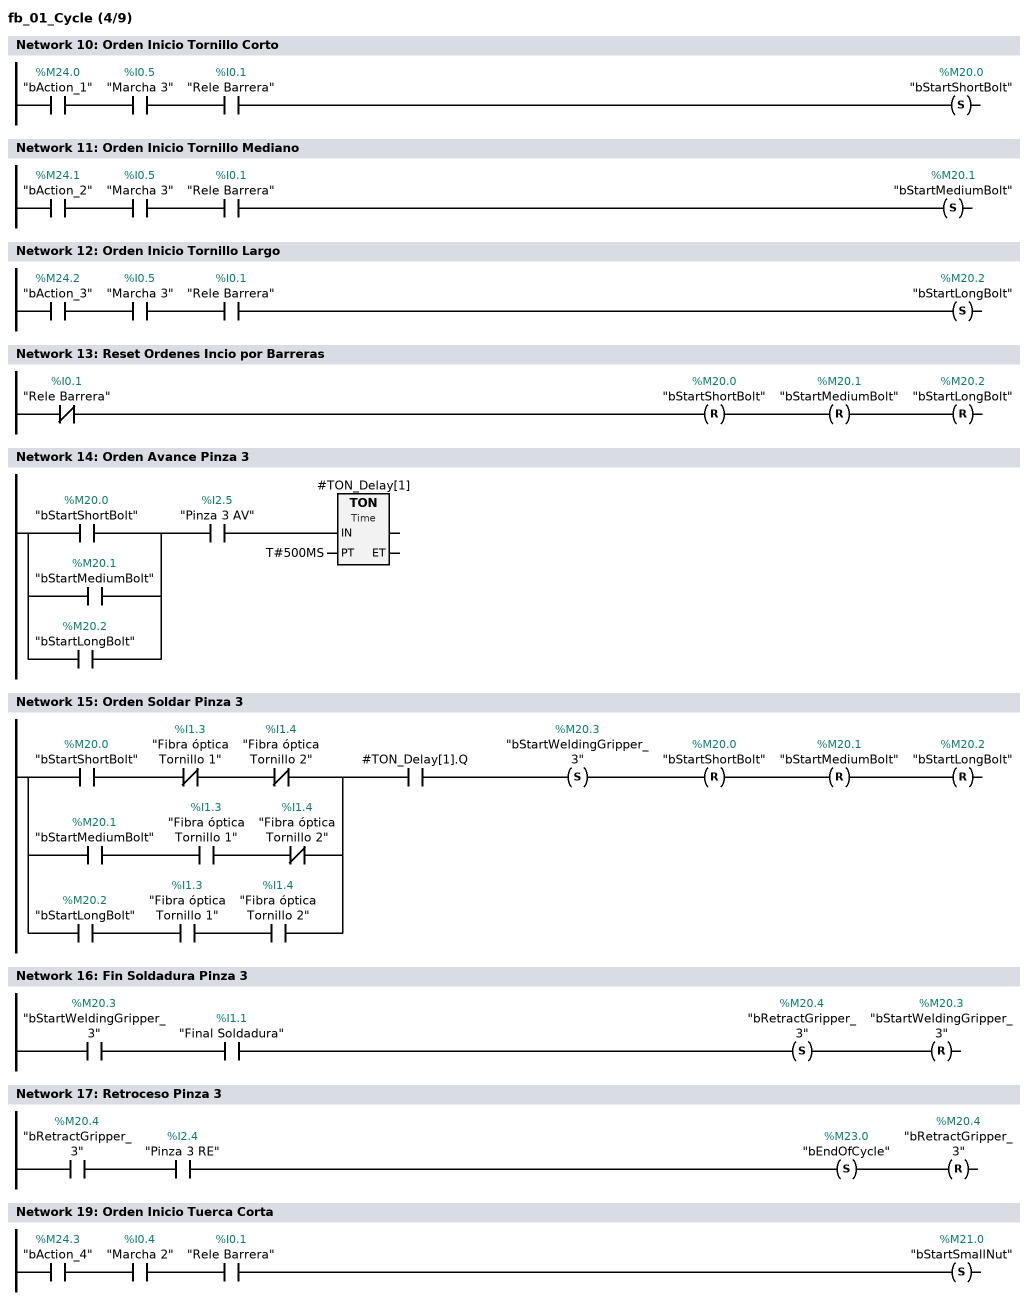
   RUNG wire#powerrail
      Contact( "bAction_1" )
      Contact( "Marcha 3" )
      Contact( "Rele Barrera" )
      S_Coil( "bStartShortBolt" )
   END_RUNG
   // the same network as SCL:
   IF "bAction_1" AND "Marcha 3" AND "Rele Barrera" THEN "bStartShortBolt" := TRUE; END_IF;
END_REGION

REGION Network 11: Orden Inicio Tornillo Mediano
   RUNG wire#powerrail
      Contact( "bAction_2" )
      Contact( "Marcha 3" )
      Contact( "Rele Barrera" )
      S_Coil( "bStartMediumBolt" )
   END_RUNG
   // the same network as SCL:
   IF "bAction_2" AND "Marcha 3" AND "Rele Barrera" THEN "bStartMediumBolt" := TRUE; END_IF;
END_REGION

REGION Network 12: Orden Inicio Tornillo Largo
   RUNG wire#powerrail
      Contact( "bAction_3" )
      Contact( "Marcha 3" )
      Contact( "Rele Barrera" )
      S_Coil( "bStartLongBolt" )
   END_RUNG
   // the same network as SCL:
   IF "bAction_3" AND "Marcha 3" AND "Rele Barrera" THEN "bStartLongBolt" := TRUE; END_IF;
END_REGION

REGION Network 13: Reset Ordenes Incio por Barreras
   RUNG wire#powerrail
      I_Contact( "Rele Barrera" )
      R_Coil( "bStartShortBolt" )
      R_Coil( "bStartMediumBolt" )
      R_Coil( "bStartLongBolt" )
   END_RUNG
   // the same network as SCL:
   IF NOT "Rele Barrera" THEN
       "bStartShortBolt" := FALSE;
       "bStartMediumBolt" := FALSE;
       "bStartLongBolt" := FALSE;
   END_IF;
END_REGION

REGION Network 14: Orden Avance Pinza 3
   RUNG wire#powerrail
      Contact( "bStartShortBolt" )
      wire#w1
      Contact( "Pinza 3 AV" )
      { S7_Templates := "time_type := Time" } #TON_Delay[1].TON(pt := T#500MS, et =>)
   END_RUNG
   RUNG wire#powerrail
      Contact( "bStartMediumBolt" )
   END_RUNG wire#w1
   RUNG wire#powerrail
      Contact( "bStartLongBolt" )
   END_RUNG wire#w1
   // the same network as SCL:
   #TON_Delay[1].TON(IN := ("bStartShortBolt" OR "bStartMediumBolt" OR "bStartLongBolt") AND "Pinza 3 AV",
                     PT := T#500MS);
END_REGION

REGION Network 15: Orden Soldar Pinza 3
   RUNG wire#powerrail
      Contact( "bStartShortBolt" )
      I_Contact( "Fibra óptica Tornillo 1" )
      I_Contact( "Fibra óptica Tornillo 2" )
      wire#w1
      Contact( #TON_Delay[1].Q )
      S_Coil( "bStartWeldingGripper_3" )
      R_Coil( "bStartShortBolt" )
      R_Coil( "bStartMediumBolt" )
      R_Coil( "bStartLongBolt" )
   END_RUNG
   RUNG wire#powerrail
      Contact( "bStartMediumBolt" )
      Contact( "Fibra óptica Tornillo 1" )
      I_Contact( "Fibra óptica Tornillo 2" )
   END_RUNG wire#w1
   RUNG wire#powerrail
      Contact( "bStartLongBolt" )
      Contact( "Fibra óptica Tornillo 1" )
      Contact( "Fibra óptica Tornillo 2" )
   END_RUNG wire#w1
   // the same network as SCL:
   IF (("bStartShortBolt" AND NOT "Fibra óptica Tornillo 1" AND NOT "Fibra óptica Tornillo 2") OR ("bStartMediumBolt" AND "Fibra óptica Tornillo 1" AND NOT "Fibra óptica Tornillo 2") OR ("bStartLongBolt" AND "Fibra óptica Tornillo 1" AND "Fibra óptica Tornillo 2")) AND #TON_Delay[1].Q THEN
       "bStartWeldingGripper_3" := TRUE;
   END_IF;
   #_w1 := (("bStartShortBolt" AND NOT "Fibra óptica Tornillo 1" AND NOT "Fibra óptica Tornillo 2") OR ("bStartMediumBolt" AND "Fibra óptica Tornillo 1" AND NOT "Fibra óptica Tornillo 2") OR ("bStartLongBolt" AND "Fibra óptica Tornillo 1" AND "Fibra óptica Tornillo 2")) AND #TON_Delay[1].Q;
   IF #_w1 THEN
       "bStartShortBolt" := FALSE;
       "bStartMediumBolt" := FALSE;
       "bStartLongBolt" := FALSE;
   END_IF;
END_REGION

REGION Network 16: Fin Soldadura Pinza 3
   RUNG wire#powerrail
      Contact( "bStartWeldingGripper_3" )
      Contact( "Final Soldadura" )
      S_Coil( "bRetractGripper_3" )
      R_Coil( "bStartWeldingGripper_3" )
   END_RUNG
   // the same network as SCL:
   IF "bStartWeldingGripper_3" AND "Final Soldadura" THEN
       "bRetractGripper_3" := TRUE;
       "bStartWeldingGripper_3" := FALSE;
   END_IF;
END_REGION

REGION Network 17: Retroceso Pinza 3
   RUNG wire#powerrail
      Contact( "bRetractGripper_3" )
      Contact( "Pinza 3 RE" )
      S_Coil( "bEndOfCycle" )
      R_Coil( "bRetractGripper_3" )
   END_RUNG
   // the same network as SCL:
   IF "bRetractGripper_3" AND "Pinza 3 RE" THEN
       "bEndOfCycle" := TRUE;
       "bRetractGripper_3" := FALSE;
   END_IF;
END_REGION

REGION Network 19: Orden Inicio Tuerca Corta
   RUNG wire#powerrail
      Contact( "bAction_4" )
      Contact( "Marcha 2" )
      Contact( "Rele Barrera" )
      S_Coil( "bStartSmallNut" )
   END_RUNG
   // the same network as SCL:
   IF "bAction_4" AND "Marcha 2" AND "Rele Barrera" THEN "bStartSmallNut" := TRUE; END_IF;
END_REGION

REGION Network 20: Orden Inicio Tuerca Larga
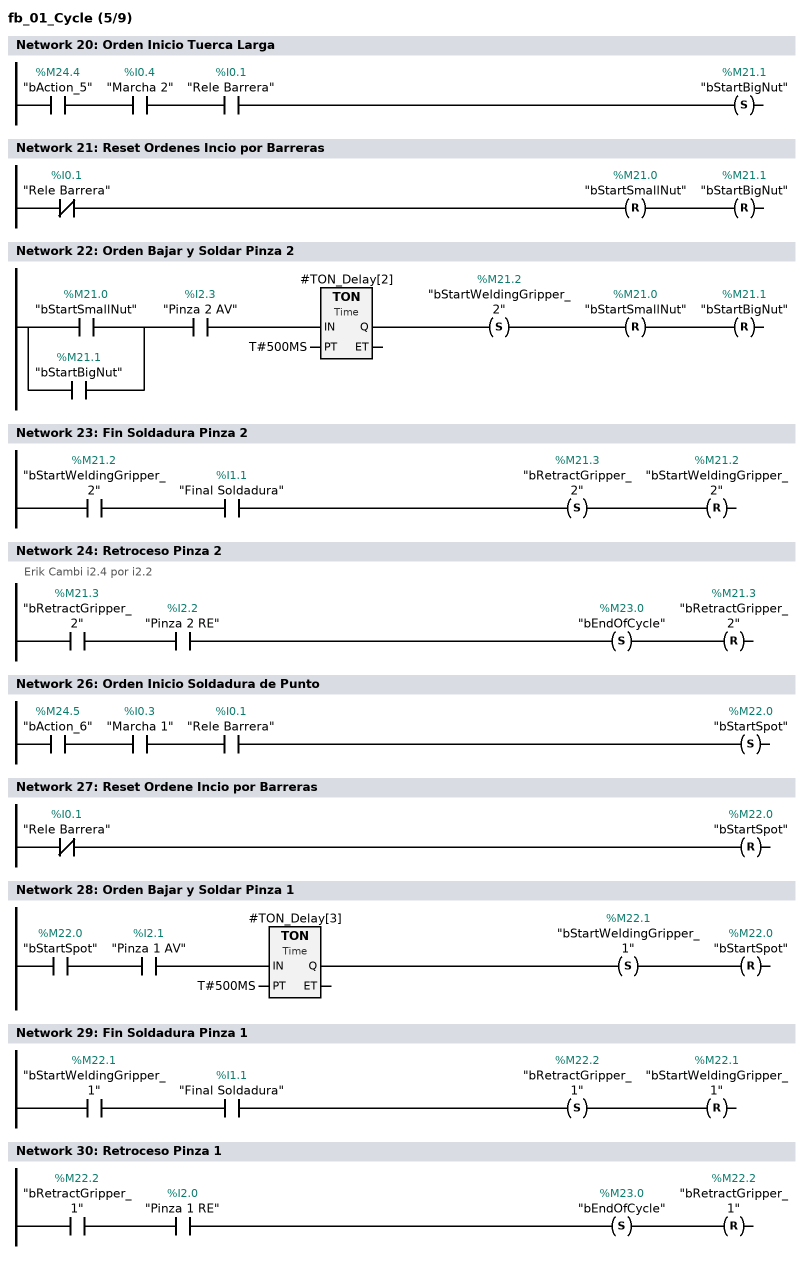
   RUNG wire#powerrail
      Contact( "bAction_5" )
      Contact( "Marcha 2" )
      Contact( "Rele Barrera" )
      S_Coil( "bStartBigNut" )
   END_RUNG
   // the same network as SCL:
   IF "bAction_5" AND "Marcha 2" AND "Rele Barrera" THEN "bStartBigNut" := TRUE; END_IF;
END_REGION

REGION Network 21: Reset Ordenes Incio por Barreras
   RUNG wire#powerrail
      I_Contact( "Rele Barrera" )
      R_Coil( "bStartSmallNut" )
      R_Coil( "bStartBigNut" )
   END_RUNG
   // the same network as SCL:
   IF NOT "Rele Barrera" THEN
       "bStartSmallNut" := FALSE;
       "bStartBigNut" := FALSE;
   END_IF;
END_REGION

REGION Network 22: Orden Bajar y Soldar Pinza 2
   RUNG wire#powerrail
      Contact( "bStartSmallNut" )
      wire#w1
      Contact( "Pinza 2 AV" )
      { S7_Templates := "time_type := Time" } #TON_Delay[2].TON(pt := T#500MS, et =>)
      S_Coil( "bStartWeldingGripper_2" )
      R_Coil( "bStartSmallNut" )
      R_Coil( "bStartBigNut" )
   END_RUNG
   RUNG wire#powerrail
      Contact( "bStartBigNut" )
   END_RUNG wire#w1
   // the same network as SCL:
   #TON_Delay[2].TON(IN := ("bStartSmallNut" OR "bStartBigNut") AND "Pinza 2 AV", PT := T#500MS);
   IF #TON_Delay[2].Q THEN
       "bStartWeldingGripper_2" := TRUE;
       "bStartSmallNut" := FALSE;
       "bStartBigNut" := FALSE;
   END_IF;
END_REGION

REGION Network 23: Fin Soldadura Pinza 2
   RUNG wire#powerrail
      Contact( "bStartWeldingGripper_2" )
      Contact( "Final Soldadura" )
      S_Coil( "bRetractGripper_2" )
      R_Coil( "bStartWeldingGripper_2" )
   END_RUNG
   // the same network as SCL:
   IF "bStartWeldingGripper_2" AND "Final Soldadura" THEN
       "bRetractGripper_2" := TRUE;
       "bStartWeldingGripper_2" := FALSE;
   END_IF;
END_REGION

REGION Network 24: Retroceso Pinza 2
   // Erik Cambi i2.4 por i2.2
   RUNG wire#powerrail
      Contact( "bRetractGripper_2" )
      Contact( "Pinza 2 RE" )
      S_Coil( "bEndOfCycle" )
      R_Coil( "bRetractGripper_2" )
   END_RUNG
   // the same network as SCL:
   IF "bRetractGripper_2" AND "Pinza 2 RE" THEN
       "bEndOfCycle" := TRUE;
       "bRetractGripper_2" := FALSE;
   END_IF;
END_REGION

REGION Network 26: Orden Inicio Soldadura de Punto
   RUNG wire#powerrail
      Contact( "bAction_6" )
      Contact( "Marcha 1" )
      Contact( "Rele Barrera" )
      S_Coil( "bStartSpot" )
   END_RUNG
   // the same network as SCL:
   IF "bAction_6" AND "Marcha 1" AND "Rele Barrera" THEN "bStartSpot" := TRUE; END_IF;
END_REGION

REGION Network 27: Reset Ordene Incio por Barreras
   RUNG wire#powerrail
      I_Contact( "Rele Barrera" )
      R_Coil( "bStartSpot" )
   END_RUNG
   // the same network as SCL:
   IF NOT "Rele Barrera" THEN "bStartSpot" := FALSE; END_IF;
END_REGION

REGION Network 28: Orden Bajar y Soldar Pinza 1
   RUNG wire#powerrail
      Contact( "bStartSpot" )
      Contact( "Pinza 1 AV" )
      { S7_Templates := "time_type := Time" } #TON_Delay[3].TON(pt := T#500MS, et =>)
      S_Coil( "bStartWeldingGripper_1" )
      R_Coil( "bStartSpot" )
   END_RUNG
   // the same network as SCL:
   #TON_Delay[3].TON(IN := "bStartSpot" AND "Pinza 1 AV", PT := T#500MS);
   IF #TON_Delay[3].Q THEN
       "bStartWeldingGripper_1" := TRUE;
       "bStartSpot" := FALSE;
   END_IF;
END_REGION

REGION Network 29: Fin Soldadura Pinza 1
   RUNG wire#powerrail
      Contact( "bStartWeldingGripper_1" )
      Contact( "Final Soldadura" )
      S_Coil( "bRetractGripper_1" )
      R_Coil( "bStartWeldingGripper_1" )
   END_RUNG
   // the same network as SCL:
   IF "bStartWeldingGripper_1" AND "Final Soldadura" THEN
       "bRetractGripper_1" := TRUE;
       "bStartWeldingGripper_1" := FALSE;
   END_IF;
END_REGION

REGION Network 30: Retroceso Pinza 1
   RUNG wire#powerrail
      Contact( "bRetractGripper_1" )
      Contact( "Pinza 1 RE" )
      S_Coil( "bEndOfCycle" )
      R_Coil( "bRetractGripper_1" )
   END_RUNG
   // the same network as SCL:
   IF "bRetractGripper_1" AND "Pinza 1 RE" THEN
       "bEndOfCycle" := TRUE;
       "bRetractGripper_1" := FALSE;
   END_IF;
END_REGION

REGION Network 32: Pieza Mala Por Soldadura
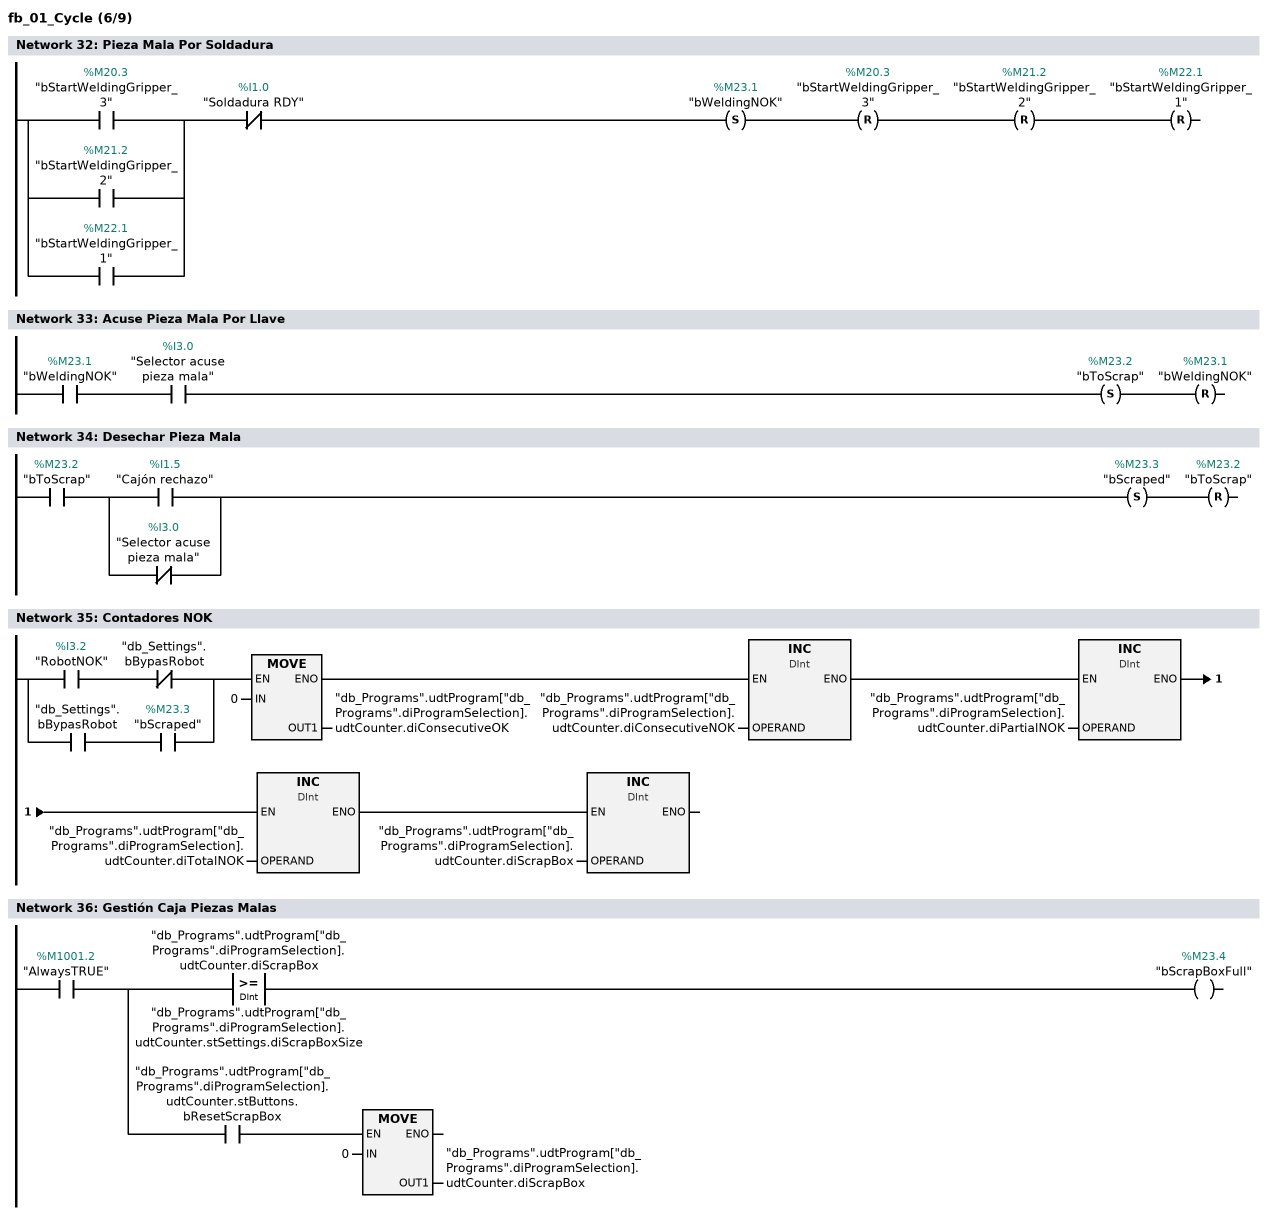
   RUNG wire#powerrail
      Contact( "bStartWeldingGripper_3" )
      wire#w1
      I_Contact( "Soldadura RDY" )
      S_Coil( "bWeldingNOK" )
      R_Coil( "bStartWeldingGripper_3" )
      R_Coil( "bStartWeldingGripper_2" )
      R_Coil( "bStartWeldingGripper_1" )
   END_RUNG
   RUNG wire#powerrail
      Contact( "bStartWeldingGripper_2" )
   END_RUNG wire#w1
   RUNG wire#powerrail
      Contact( "bStartWeldingGripper_1" )
   END_RUNG wire#w1
   // the same network as SCL:
   IF ("bStartWeldingGripper_3" OR "bStartWeldingGripper_2" OR "bStartWeldingGripper_1") AND NOT "Soldadura RDY" THEN
       "bWeldingNOK" := TRUE;
   END_IF;
   #_w1 := ("bStartWeldingGripper_3" OR "bStartWeldingGripper_2" OR "bStartWeldingGripper_1") AND NOT "Soldadura RDY";
   IF #_w1 THEN
       "bStartWeldingGripper_3" := FALSE;
       "bStartWeldingGripper_2" := FALSE;
       "bStartWeldingGripper_1" := FALSE;
   END_IF;
END_REGION

REGION Network 33: Acuse Pieza Mala Por Llave
   RUNG wire#powerrail
      Contact( "bWeldingNOK" )
      Contact( "Selector acuse pieza mala" )
      S_Coil( "bToScrap" )
      R_Coil( "bWeldingNOK" )
   END_RUNG
   // the same network as SCL:
   IF "bWeldingNOK" AND "Selector acuse pieza mala" THEN
       "bToScrap" := TRUE;
       "bWeldingNOK" := FALSE;
   END_IF;
END_REGION

REGION Network 34: Desechar Pieza Mala
   RUNG wire#powerrail
      Contact( "bToScrap" )
      wire#w1
      Contact( "Cajón rechazo" )
      wire#w2
      S_Coil( "bScraped" )
      R_Coil( "bToScrap" )
   END_RUNG
   RUNG wire#w1
      I_Contact( "Selector acuse pieza mala" )
   END_RUNG wire#w2
   // the same network as SCL:
   IF "bToScrap" AND ("Cajón rechazo" OR NOT "Selector acuse pieza mala") THEN
       "bScraped" := TRUE;
       "bToScrap" := FALSE;
   END_IF;
END_REGION

REGION Network 35: Contadores NOK
   RUNG wire#powerrail
      Contact( "RobotNOK" )
      I_Contact( "db_Settings".bBypasRobot )
      wire#w1
      Move(in := 0, out1 => "db_Programs".udtProgram["db_Programs".diProgramSelection].udtCounter.diConsecutiveOK)
      { S7_Templates := "DestType := DInt" } Inc( "db_Programs".udtProgram["db_Programs".diProgramSelection].udtCounter.diConsecutiveNOK )
      { S7_Templates := "DestType := DInt" } Inc( "db_Programs".udtProgram["db_Programs".diProgramSelection].udtCounter.diPartialNOK )
      { S7_Templates := "DestType := DInt" } Inc( "db_Programs".udtProgram["db_Programs".diProgramSelection].udtCounter.diTotalNOK )
      { S7_Templates := "DestType := DInt" } Inc( "db_Programs".udtProgram["db_Programs".diProgramSelection].udtCounter.diScrapBox )
   END_RUNG
   RUNG wire#powerrail
      Contact( "db_Settings".bBypasRobot )
      Contact( "bScraped" )
   END_RUNG wire#w1
   // the same network as SCL:
   IF ("RobotNOK" AND NOT "db_Settings".bBypasRobot) OR ("db_Settings".bBypasRobot AND "bScraped") THEN
       "db_Programs".udtProgram["db_Programs".diProgramSelection].udtCounter.diConsecutiveOK := 0;
       "db_Programs".udtProgram["db_Programs".diProgramSelection].udtCounter.diConsecutiveNOK := "db_Programs".udtProgram["db_Programs".diProgramSelection].udtCounter.diConsecutiveNOK + 1;
       "db_Programs".udtProgram["db_Programs".diProgramSelection].udtCounter.diPartialNOK := "db_Programs".udtProgram["db_Programs".diProgramSelection].udtCounter.diPartialNOK + 1;
       "db_Programs".udtProgram["db_Programs".diProgramSelection].udtCounter.diTotalNOK := "db_Programs".udtProgram["db_Programs".diProgramSelection].udtCounter.diTotalNOK + 1;
       "db_Programs".udtProgram["db_Programs".diProgramSelection].udtCounter.diScrapBox := "db_Programs".udtProgram["db_Programs".diProgramSelection].udtCounter.diScrapBox + 1;
   END_IF;
END_REGION

REGION Network 36: Gestión Caja Piezas Malas
   RUNG wire#powerrail
      Contact( "AlwaysTRUE" )
      wire#w1
      { S7_Templates := "SrcType := DInt" } GE_Contact(in1 := "db_Programs".udtProgram["db_Programs".diProgramSelection].udtCounter.diScrapBox, in2 := "db_Programs".udtProgram["db_Programs".diProgramSelection].udtCounter.stSettings.diScrapBoxSize)
      Coil( "bScrapBoxFull" )
   END_RUNG
   RUNG wire#w1
      Contact( "db_Programs".udtProgram["db_Programs".diProgramSelection].udtCounter.stButtons.bResetScrapBox )
      Move(in := 0, out1 => "db_Programs".udtProgram["db_Programs".diProgramSelection].udtCounter.diScrapBox)
   END_RUNG
   // the same network as SCL:
   "bScrapBoxFull" := "AlwaysTRUE" AND ("db_Programs".udtProgram["db_Programs".diProgramSelection].udtCounter.diScrapBox >= "db_Programs".udtProgram["db_Programs".diProgramSelection].udtCounter.stSettings.diScrapBoxSize);
   IF "AlwaysTRUE" AND "db_Programs".udtProgram["db_Programs".diProgramSelection].udtCounter.stButtons.bResetScrapBox THEN
       "db_Programs".udtProgram["db_Programs".diProgramSelection].udtCounter.diScrapBox := 0;
   END_IF;
END_REGION

REGION Network 37: Gestión Contadores NOK
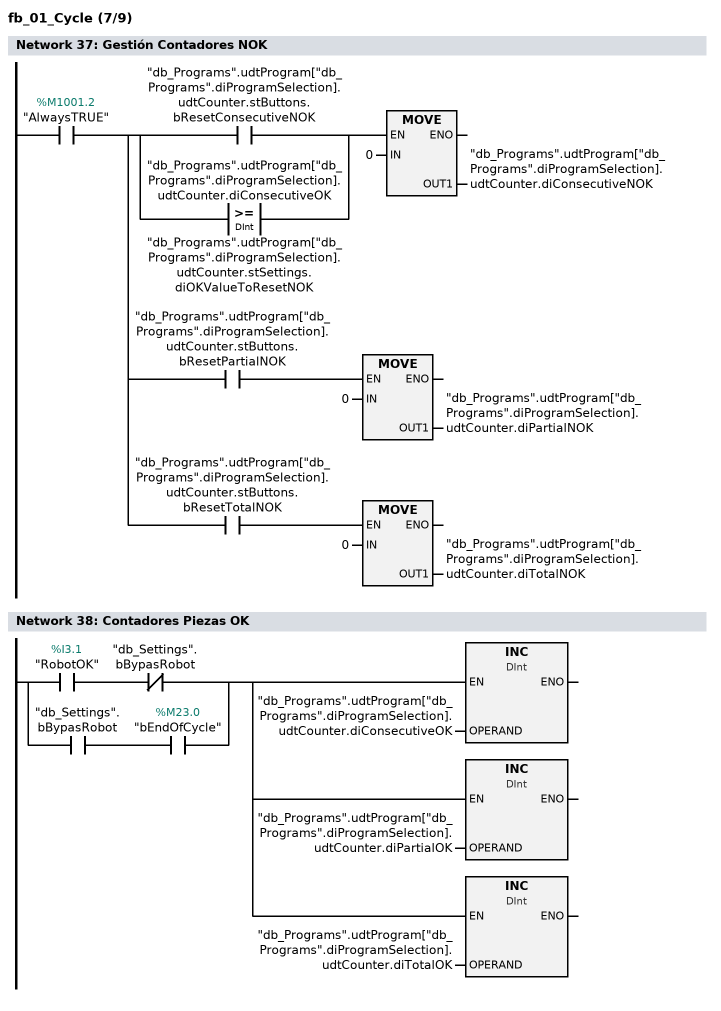
   RUNG wire#powerrail
      Contact( "AlwaysTRUE" )
      wire#w1
      Contact( "db_Programs".udtProgram["db_Programs".diProgramSelection].udtCounter.stButtons.bResetConsecutiveNOK )
      wire#w2
      Move(in := 0, out1 => "db_Programs".udtProgram["db_Programs".diProgramSelection].udtCounter.diConsecutiveNOK)
   END_RUNG
   RUNG wire#w1
      { S7_Templates := "SrcType := DInt" } GE_Contact(in1 := "db_Programs".udtProgram["db_Programs".diProgramSelection].udtCounter.diConsecutiveOK, in2 := "db_Programs".udtProgram["db_Programs".diProgramSelection].udtCounter.stSettings.diOKValueToResetNOK)
   END_RUNG wire#w2
   RUNG wire#w1
      Contact( "db_Programs".udtProgram["db_Programs".diProgramSelection].udtCounter.stButtons.bResetPartialNOK )
      Move(in := 0, out1 => "db_Programs".udtProgram["db_Programs".diProgramSelection].udtCounter.diPartialNOK)
   END_RUNG
   RUNG wire#w1
      Contact( "db_Programs".udtProgram["db_Programs".diProgramSelection].udtCounter.stButtons.bResetTotalNOK )
      Move(in := 0, out1 => "db_Programs".udtProgram["db_Programs".diProgramSelection].udtCounter.diTotalNOK)
   END_RUNG
   // the same network as SCL:
   IF "AlwaysTRUE" AND ("db_Programs".udtProgram["db_Programs".diProgramSelection].udtCounter.stButtons.bResetConsecutiveNOK OR ("db_Programs".udtProgram["db_Programs".diProgramSelection].udtCounter.diConsecutiveOK >= "db_Programs".udtProgram["db_Programs".diProgramSelection].udtCounter.stSettings.diOKValueToResetNOK)) THEN
       "db_Programs".udtProgram["db_Programs".diProgramSelection].udtCounter.diConsecutiveNOK := 0;
   END_IF;
   IF "AlwaysTRUE" AND "db_Programs".udtProgram["db_Programs".diProgramSelection].udtCounter.stButtons.bResetPartialNOK THEN
       "db_Programs".udtProgram["db_Programs".diProgramSelection].udtCounter.diPartialNOK := 0;
   END_IF;
   IF "AlwaysTRUE" AND "db_Programs".udtProgram["db_Programs".diProgramSelection].udtCounter.stButtons.bResetTotalNOK THEN
       "db_Programs".udtProgram["db_Programs".diProgramSelection].udtCounter.diTotalNOK := 0;
   END_IF;
END_REGION

REGION Network 38: Contadores Piezas OK
   RUNG wire#powerrail
      Contact( "RobotOK" )
      I_Contact( "db_Settings".bBypasRobot )
      wire#w1
      { S7_Templates := "DestType := DInt" } Inc( "db_Programs".udtProgram["db_Programs".diProgramSelection].udtCounter.diConsecutiveOK )
   END_RUNG
   RUNG wire#powerrail
      Contact( "db_Settings".bBypasRobot )
      Contact( "bEndOfCycle" )
   END_RUNG wire#w1
   RUNG wire#w1
      { S7_Templates := "DestType := DInt" } Inc( "db_Programs".udtProgram["db_Programs".diProgramSelection].udtCounter.diPartialOK )
   END_RUNG
   RUNG wire#w1
      { S7_Templates := "DestType := DInt" } Inc( "db_Programs".udtProgram["db_Programs".diProgramSelection].udtCounter.diTotalOK )
   END_RUNG
   // the same network as SCL:
   IF ("RobotOK" AND NOT "db_Settings".bBypasRobot) OR ("db_Settings".bBypasRobot AND "bEndOfCycle") THEN
       "db_Programs".udtProgram["db_Programs".diProgramSelection].udtCounter.diConsecutiveOK := "db_Programs".udtProgram["db_Programs".diProgramSelection].udtCounter.diConsecutiveOK + 1;
       "db_Programs".udtProgram["db_Programs".diProgramSelection].udtCounter.diPartialOK := "db_Programs".udtProgram["db_Programs".diProgramSelection].udtCounter.diPartialOK + 1;
       "db_Programs".udtProgram["db_Programs".diProgramSelection].udtCounter.diTotalOK := "db_Programs".udtProgram["db_Programs".diProgramSelection].udtCounter.diTotalOK + 1;
   END_IF;
END_REGION

REGION Network 39: Gestión Contadores OK
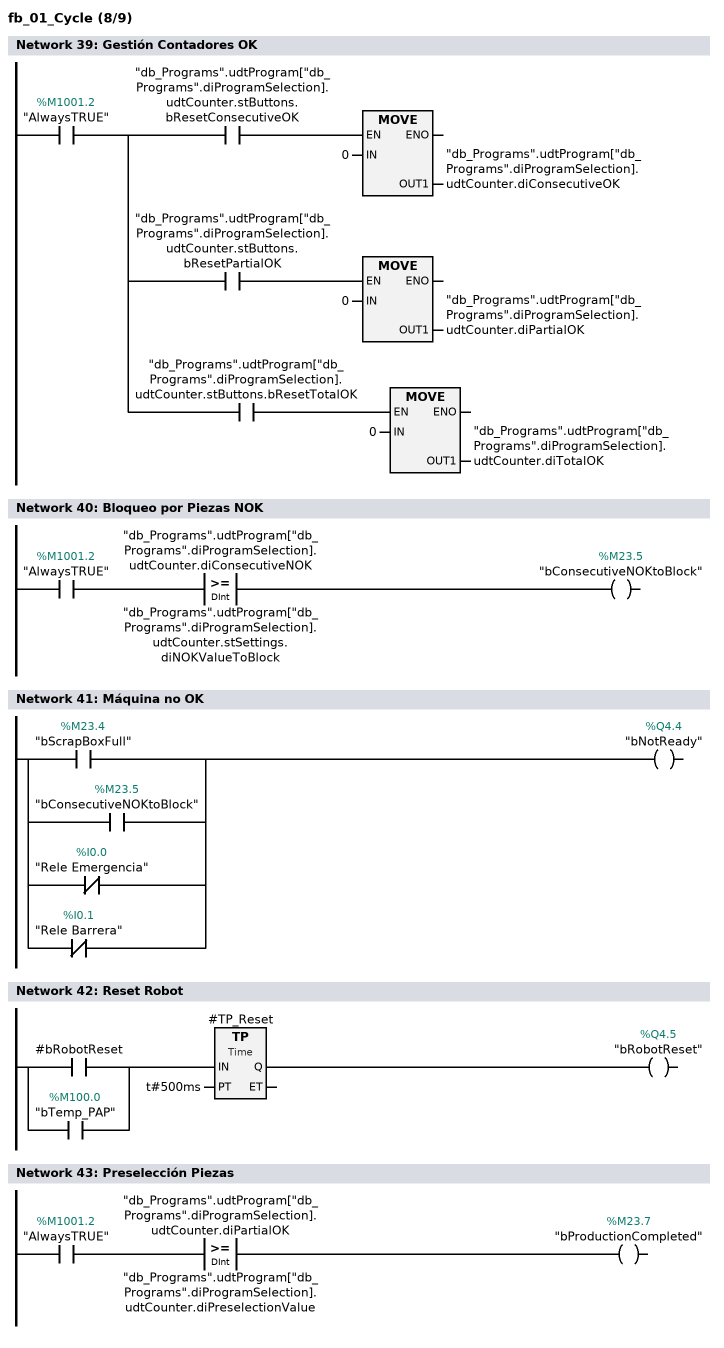
   RUNG wire#powerrail
      Contact( "AlwaysTRUE" )
      wire#w1
      Contact( "db_Programs".udtProgram["db_Programs".diProgramSelection].udtCounter.stButtons.bResetConsecutiveOK )
      Move(in := 0, out1 => "db_Programs".udtProgram["db_Programs".diProgramSelection].udtCounter.diConsecutiveOK)
   END_RUNG
   RUNG wire#w1
      Contact( "db_Programs".udtProgram["db_Programs".diProgramSelection].udtCounter.stButtons.bResetPartialOK )
      Move(in := 0, out1 => "db_Programs".udtProgram["db_Programs".diProgramSelection].udtCounter.diPartialOK)
   END_RUNG
   RUNG wire#w1
      Contact( "db_Programs".udtProgram["db_Programs".diProgramSelection].udtCounter.stButtons.bResetTotalOK )
      Move(in := 0, out1 => "db_Programs".udtProgram["db_Programs".diProgramSelection].udtCounter.diTotalOK)
   END_RUNG
   // the same network as SCL:
   IF "AlwaysTRUE" AND "db_Programs".udtProgram["db_Programs".diProgramSelection].udtCounter.stButtons.bResetConsecutiveOK THEN
       "db_Programs".udtProgram["db_Programs".diProgramSelection].udtCounter.diConsecutiveOK := 0;
   END_IF;
   IF "AlwaysTRUE" AND "db_Programs".udtProgram["db_Programs".diProgramSelection].udtCounter.stButtons.bResetPartialOK THEN
       "db_Programs".udtProgram["db_Programs".diProgramSelection].udtCounter.diPartialOK := 0;
   END_IF;
   IF "AlwaysTRUE" AND "db_Programs".udtProgram["db_Programs".diProgramSelection].udtCounter.stButtons.bResetTotalOK THEN
       "db_Programs".udtProgram["db_Programs".diProgramSelection].udtCounter.diTotalOK := 0;
   END_IF;
END_REGION

REGION Network 40: Bloqueo por Piezas NOK
   RUNG wire#powerrail
      Contact( "AlwaysTRUE" )
      { S7_Templates := "SrcType := DInt" } GE_Contact(in1 := "db_Programs".udtProgram["db_Programs".diProgramSelection].udtCounter.diConsecutiveNOK, in2 := "db_Programs".udtProgram["db_Programs".diProgramSelection].udtCounter.stSettings.diNOKValueToBlock)
      Coil( "bConsecutiveNOKtoBlock" )
   END_RUNG
   // the same network as SCL:
   "bConsecutiveNOKtoBlock" := "AlwaysTRUE" AND ("db_Programs".udtProgram["db_Programs".diProgramSelection].udtCounter.diConsecutiveNOK >= "db_Programs".udtProgram["db_Programs".diProgramSelection].udtCounter.stSettings.diNOKValueToBlock);
END_REGION

REGION Network 41: Máquina no OK
   RUNG wire#powerrail
      Contact( "bScrapBoxFull" )
      wire#w1
      Coil( "bNotReady" )
   END_RUNG
   RUNG wire#powerrail
      Contact( "bConsecutiveNOKtoBlock" )
   END_RUNG wire#w1
   RUNG wire#powerrail
      I_Contact( "Rele Emergencia" )
   END_RUNG wire#w1
   RUNG wire#powerrail
      I_Contact( "Rele Barrera" )
   END_RUNG wire#w1
   // the same network as SCL:
   "bNotReady" := "bScrapBoxFull" OR "bConsecutiveNOKtoBlock" OR NOT "Rele Emergencia" OR NOT "Rele Barrera";
END_REGION

REGION Network 42: Reset Robot
   RUNG wire#powerrail
      Contact( #bRobotReset )
      wire#w1
      { S7_Templates := "time_type := Time" } #TP_Reset.TP(pt := t#500ms, et =>)
      Coil( "bRobotReset" )
   END_RUNG
   RUNG wire#powerrail
      Contact( "bTemp_PAP" )
   END_RUNG wire#w1
   // the same network as SCL:
   #TP_Reset(IN := #bRobotReset OR "bTemp_PAP", PT := t#500ms);   // TP
   "bRobotReset" := #TP_Reset.Q;
END_REGION

REGION Network 43: Preselección Piezas
   RUNG wire#powerrail
      Contact( "AlwaysTRUE" )
      { S7_Templates := "SrcType := DInt" } GE_Contact(in1 := "db_Programs".udtProgram["db_Programs".diProgramSelection].udtCounter.diPartialOK, in2 := "db_Programs".udtProgram["db_Programs".diProgramSelection].udtCounter.diPreselectionValue)
      Coil( "bProductionCompleted" )
   END_RUNG
   // the same network as SCL:
   "bProductionCompleted" := "AlwaysTRUE" AND ("db_Programs".udtProgram["db_Programs".diProgramSelection].udtCounter.diPartialOK >= "db_Programs".udtProgram["db_Programs".diProgramSelection].udtCounter.diPreselectionValue);
END_REGION

REGION Network 45: Incremento Paso de Ciclo
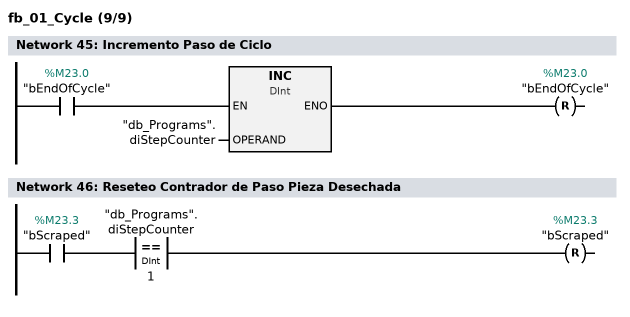
   RUNG wire#powerrail
      Contact( "bEndOfCycle" )
      { S7_Templates := "DestType := DInt" } Inc( "db_Programs".diStepCounter )
      R_Coil( "bEndOfCycle" )
   END_RUNG
   // the same network as SCL:
   IF "bEndOfCycle" THEN
       "db_Programs".diStepCounter := "db_Programs".diStepCounter + 1;
       "bEndOfCycle" := FALSE;
   END_IF;
END_REGION

REGION Network 46: Reseteo Contrador de Paso Pieza Desechada
   RUNG wire#powerrail
      Contact( "bScraped" )
      { S7_Templates := "SrcType := DInt" } EQ_Contact(in1 := "db_Programs".diStepCounter, in2 := 1)
      R_Coil( "bScraped" )
   END_RUNG
   // the same network as SCL:
   IF "bScraped" AND ("db_Programs".diStepCounter = 1) THEN "bScraped" := FALSE; END_IF;
END_REGION
END_FUNCTION_BLOCK

FUNCTION "fc_02_Outputs" : Void   // FC2, LAD
{ S7_Optimized_Access := 'TRUE' }
VERSION : 0.1
// stored: AutoNumber false, IsIECCheckEnabled false, SetENOAutomatically false, UDAEnableTagReadback false
   VAR_TEMP
      bIsInverted : Bool;
   END_VAR
   VAR_TEMP   // added for the SCL form of the ladder/FBD networks
      _w1 : Bool;
      _w2 : Bool;
      _w3 : Bool;
      _w4 : Bool;
   END_VAR
BEGIN

REGION Network 1: Rele rearme
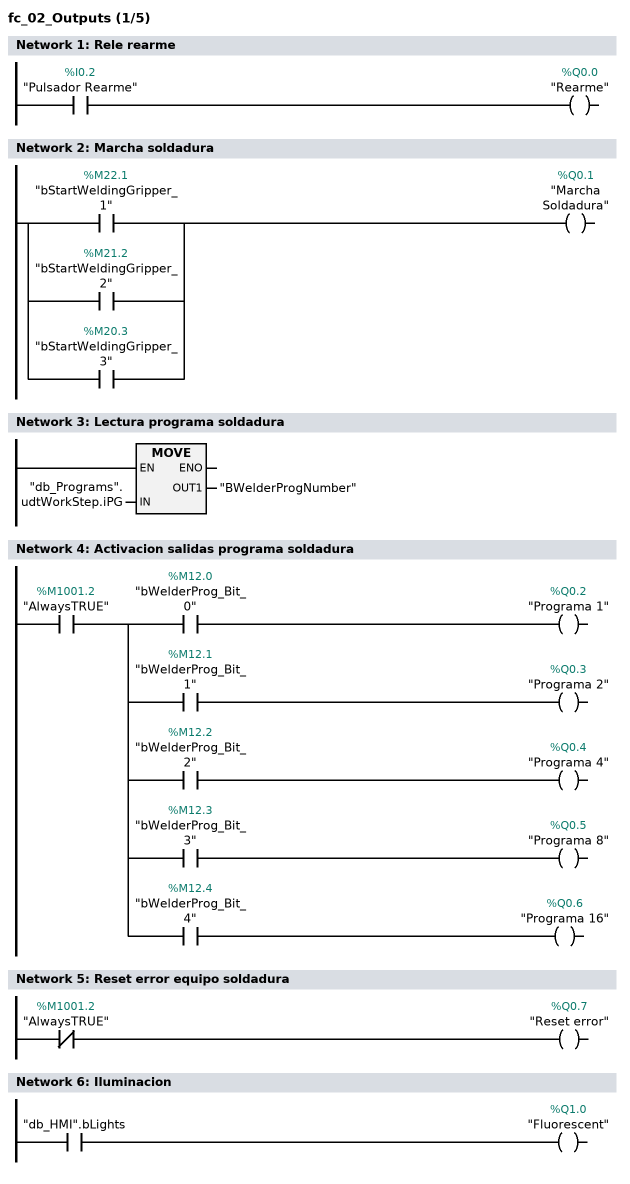
   RUNG wire#powerrail
      Contact( "Pulsador Rearme" )
      Coil( "Rearme" )
   END_RUNG
   // the same network as SCL:
   "Rearme" := "Pulsador Rearme";
END_REGION

REGION Network 2: Marcha soldadura
   RUNG wire#powerrail
      Contact( "bStartWeldingGripper_1" )
      wire#w1
      Coil( "Marcha Soldadura" )
   END_RUNG
   RUNG wire#powerrail
      Contact( "bStartWeldingGripper_2" )
   END_RUNG wire#w1
   RUNG wire#powerrail
      Contact( "bStartWeldingGripper_3" )
   END_RUNG wire#w1
   // the same network as SCL:
   "Marcha Soldadura" := "bStartWeldingGripper_1" OR "bStartWeldingGripper_2" OR "bStartWeldingGripper_3";
END_REGION

REGION Network 3: Lectura programa soldadura
   RUNG wire#powerrail
      Move(in := "db_Programs".udtWorkStep.iPG, out1 => "BWelderProgNumber")
   END_RUNG
   // the same network as SCL:
   "BWelderProgNumber" := "db_Programs".udtWorkStep.iPG;
END_REGION

REGION Network 4: Activacion salidas programa soldadura
   RUNG wire#powerrail
      Contact( "AlwaysTRUE" )
      wire#w1
      Contact( "bWelderProg_Bit_0" )
      Coil( "Programa 1" )
   END_RUNG
   RUNG wire#w1
      Contact( "bWelderProg_Bit_1" )
      Coil( "Programa 2" )
   END_RUNG
   RUNG wire#w1
      Contact( "bWelderProg_Bit_2" )
      Coil( "Programa 4" )
   END_RUNG
   RUNG wire#w1
      Contact( "bWelderProg_Bit_3" )
      Coil( "Programa 8" )
   END_RUNG
   RUNG wire#w1
      Contact( "bWelderProg_Bit_4" )
      Coil( "Programa 16" )
   END_RUNG
   // the same network as SCL:
   "Programa 1" := "AlwaysTRUE" AND "bWelderProg_Bit_0";
   "Programa 2" := "AlwaysTRUE" AND "bWelderProg_Bit_1";
   "Programa 4" := "AlwaysTRUE" AND "bWelderProg_Bit_2";
   "Programa 8" := "AlwaysTRUE" AND "bWelderProg_Bit_3";
   "Programa 16" := "AlwaysTRUE" AND "bWelderProg_Bit_4";
END_REGION

REGION Network 5: Reset error equipo soldadura
   RUNG wire#powerrail
      I_Contact( "AlwaysTRUE" )
      Coil( "Reset error" )
   END_RUNG
   // the same network as SCL:
   "Reset error" := NOT "AlwaysTRUE";
END_REGION

REGION Network 6: Iluminacion
   RUNG wire#powerrail
      Contact( "db_HMI".bLights )
      Coil( "Fluorescent" )
   END_RUNG
   // the same network as SCL:
   "Fluorescent" := "db_HMI".bLights;
END_REGION

REGION Network 7: Pilotos 1
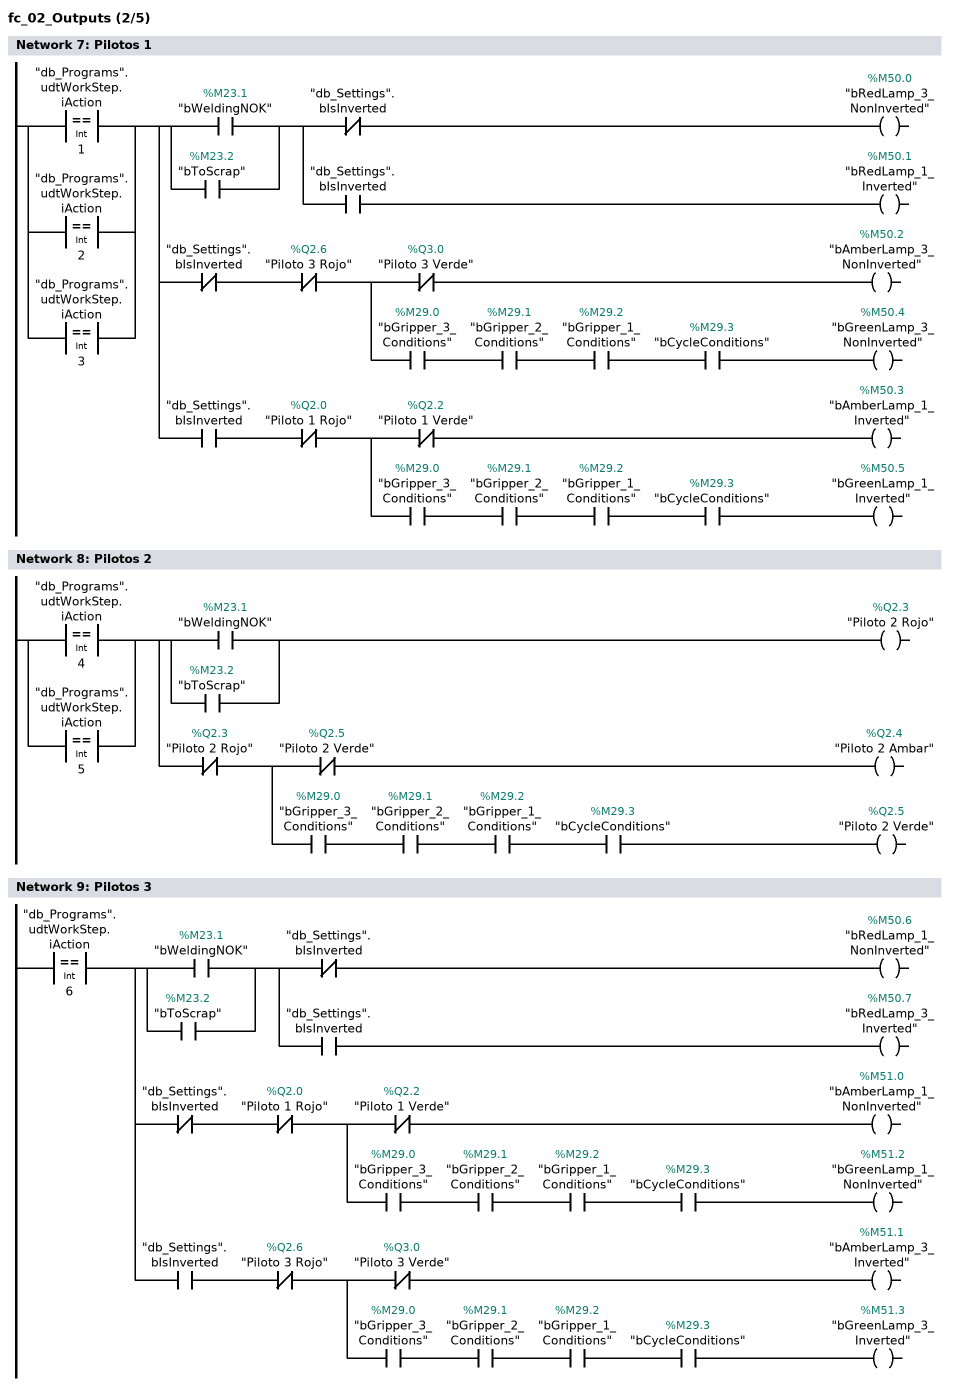
   RUNG wire#powerrail
      { S7_Templates := "SrcType := Int" } EQ_Contact(in1 := "db_Programs".udtWorkStep.iAction, in2 := 1)
      wire#w1
      Contact( "bWeldingNOK" )
      wire#w2
      I_Contact( "db_Settings".bIsInverted )
      Coil( "bRedLamp_3_NonInverted" )
   END_RUNG
   RUNG wire#powerrail
      { S7_Templates := "SrcType := Int" } EQ_Contact(in1 := "db_Programs".udtWorkStep.iAction, in2 := 2)
   END_RUNG wire#w1
   RUNG wire#powerrail
      { S7_Templates := "SrcType := Int" } EQ_Contact(in1 := "db_Programs".udtWorkStep.iAction, in2 := 3)
   END_RUNG wire#w1
   RUNG wire#w1
      Contact( "bToScrap" )
   END_RUNG wire#w2
   RUNG wire#w2
      Contact( "db_Settings".bIsInverted )
      Coil( "bRedLamp_1_Inverted" )
   END_RUNG
   RUNG wire#w1
      I_Contact( "db_Settings".bIsInverted )
      I_Contact( "Piloto 3 Rojo" )
      wire#w3
      I_Contact( "Piloto 3 Verde" )
      Coil( "bAmberLamp_3_NonInverted" )
   END_RUNG
   RUNG wire#w3
      Contact( "bGripper_3_Conditions" )
      Contact( "bGripper_2_Conditions" )
      Contact( "bGripper_1_Conditions" )
      Contact( "bCycleConditions" )
      Coil( "bGreenLamp_3_NonInverted" )
   END_RUNG
   RUNG wire#w1
      Contact( "db_Settings".bIsInverted )
      I_Contact( "Piloto 1 Rojo" )
      wire#w4
      I_Contact( "Piloto 1 Verde" )
      Coil( "bAmberLamp_1_Inverted" )
   END_RUNG
   RUNG wire#w4
      Contact( "bGripper_3_Conditions" )
      Contact( "bGripper_2_Conditions" )
      Contact( "bGripper_1_Conditions" )
      Contact( "bCycleConditions" )
      Coil( "bGreenLamp_1_Inverted" )
   END_RUNG
   // the same network as SCL:
   #_w1 := ("db_Programs".udtWorkStep.iAction = 1) OR ("db_Programs".udtWorkStep.iAction = 2) OR ("db_Programs".udtWorkStep.iAction = 3);
   #_w2 := #_w1 AND ("bWeldingNOK" OR "bToScrap");
   "bRedLamp_3_NonInverted" := #_w2 AND NOT "db_Settings".bIsInverted;
   "bRedLamp_1_Inverted" := #_w2 AND "db_Settings".bIsInverted;
   #_w3 := #_w1 AND NOT "db_Settings".bIsInverted AND NOT "Piloto 3 Rojo";
   "bAmberLamp_3_NonInverted" := #_w3 AND NOT "Piloto 3 Verde";
   "bGreenLamp_3_NonInverted" := #_w3 AND "bGripper_3_Conditions" AND "bGripper_2_Conditions" AND "bGripper_1_Conditions" AND "bCycleConditions";
   #_w4 := #_w1 AND "db_Settings".bIsInverted AND NOT "Piloto 1 Rojo";
   "bAmberLamp_1_Inverted" := #_w4 AND NOT "Piloto 1 Verde";
   "bGreenLamp_1_Inverted" := #_w4 AND "bGripper_3_Conditions" AND "bGripper_2_Conditions" AND "bGripper_1_Conditions" AND "bCycleConditions";
END_REGION

REGION Network 8: Pilotos 2
   RUNG wire#powerrail
      { S7_Templates := "SrcType := Int" } EQ_Contact(in1 := "db_Programs".udtWorkStep.iAction, in2 := 4)
      wire#w1
      Contact( "bWeldingNOK" )
      wire#w2
      Coil( "Piloto 2 Rojo" )
   END_RUNG
   RUNG wire#powerrail
      { S7_Templates := "SrcType := Int" } EQ_Contact(in1 := "db_Programs".udtWorkStep.iAction, in2 := 5)
   END_RUNG wire#w1
   RUNG wire#w1
      Contact( "bToScrap" )
   END_RUNG wire#w2
   RUNG wire#w1
      I_Contact( "Piloto 2 Rojo" )
      wire#w3
      I_Contact( "Piloto 2 Verde" )
      Coil( "Piloto 2 Ambar" )
   END_RUNG
   RUNG wire#w3
      Contact( "bGripper_3_Conditions" )
      Contact( "bGripper_2_Conditions" )
      Contact( "bGripper_1_Conditions" )
      Contact( "bCycleConditions" )
      Coil( "Piloto 2 Verde" )
   END_RUNG
   // the same network as SCL:
   #_w1 := ("db_Programs".udtWorkStep.iAction = 4) OR ("db_Programs".udtWorkStep.iAction = 5);
   "Piloto 2 Rojo" := #_w1 AND ("bWeldingNOK" OR "bToScrap");
   #_w2 := #_w1 AND NOT "Piloto 2 Rojo";
   "Piloto 2 Ambar" := #_w2 AND NOT "Piloto 2 Verde";
   "Piloto 2 Verde" := #_w2 AND "bGripper_3_Conditions" AND "bGripper_2_Conditions" AND "bGripper_1_Conditions" AND "bCycleConditions";
END_REGION

REGION Network 9: Pilotos 3
   RUNG wire#powerrail
      { S7_Templates := "SrcType := Int" } EQ_Contact(in1 := "db_Programs".udtWorkStep.iAction, in2 := 6)
      wire#w1
      Contact( "bWeldingNOK" )
      wire#w2
      I_Contact( "db_Settings".bIsInverted )
      Coil( "bRedLamp_1_NonInverted" )
   END_RUNG
   RUNG wire#w1
      Contact( "bToScrap" )
   END_RUNG wire#w2
   RUNG wire#w2
      Contact( "db_Settings".bIsInverted )
      Coil( "bRedLamp_3_Inverted" )
   END_RUNG
   RUNG wire#w1
      I_Contact( "db_Settings".bIsInverted )
      I_Contact( "Piloto 1 Rojo" )
      wire#w3
      I_Contact( "Piloto 1 Verde" )
      Coil( "bAmberLamp_1_NonInverted" )
   END_RUNG
   RUNG wire#w3
      Contact( "bGripper_3_Conditions" )
      Contact( "bGripper_2_Conditions" )
      Contact( "bGripper_1_Conditions" )
      Contact( "bCycleConditions" )
      Coil( "bGreenLamp_1_NonInverted" )
   END_RUNG
   RUNG wire#w1
      Contact( "db_Settings".bIsInverted )
      I_Contact( "Piloto 3 Rojo" )
      wire#w4
      I_Contact( "Piloto 3 Verde" )
      Coil( "bAmberLamp_3_Inverted" )
   END_RUNG
   RUNG wire#w4
      Contact( "bGripper_3_Conditions" )
      Contact( "bGripper_2_Conditions" )
      Contact( "bGripper_1_Conditions" )
      Contact( "bCycleConditions" )
      Coil( "bGreenLamp_3_Inverted" )
   END_RUNG
   // the same network as SCL:
   #_w1 := "db_Programs".udtWorkStep.iAction = 6;
   #_w2 := #_w1 AND ("bWeldingNOK" OR "bToScrap");
   "bRedLamp_1_NonInverted" := #_w2 AND NOT "db_Settings".bIsInverted;
   "bRedLamp_3_Inverted" := #_w2 AND "db_Settings".bIsInverted;
   #_w3 := #_w1 AND NOT "db_Settings".bIsInverted AND NOT "Piloto 1 Rojo";
   "bAmberLamp_1_NonInverted" := #_w3 AND NOT "Piloto 1 Verde";
   "bGreenLamp_1_NonInverted" := #_w3 AND "bGripper_3_Conditions" AND "bGripper_2_Conditions" AND "bGripper_1_Conditions" AND "bCycleConditions";
   #_w4 := #_w1 AND "db_Settings".bIsInverted AND NOT "Piloto 3 Rojo";
   "bAmberLamp_3_Inverted" := #_w4 AND NOT "Piloto 3 Verde";
   "bGreenLamp_3_Inverted" := #_w4 AND "bGripper_3_Conditions" AND "bGripper_2_Conditions" AND "bGripper_1_Conditions" AND "bCycleConditions";
END_REGION

REGION Network 10: Baliza
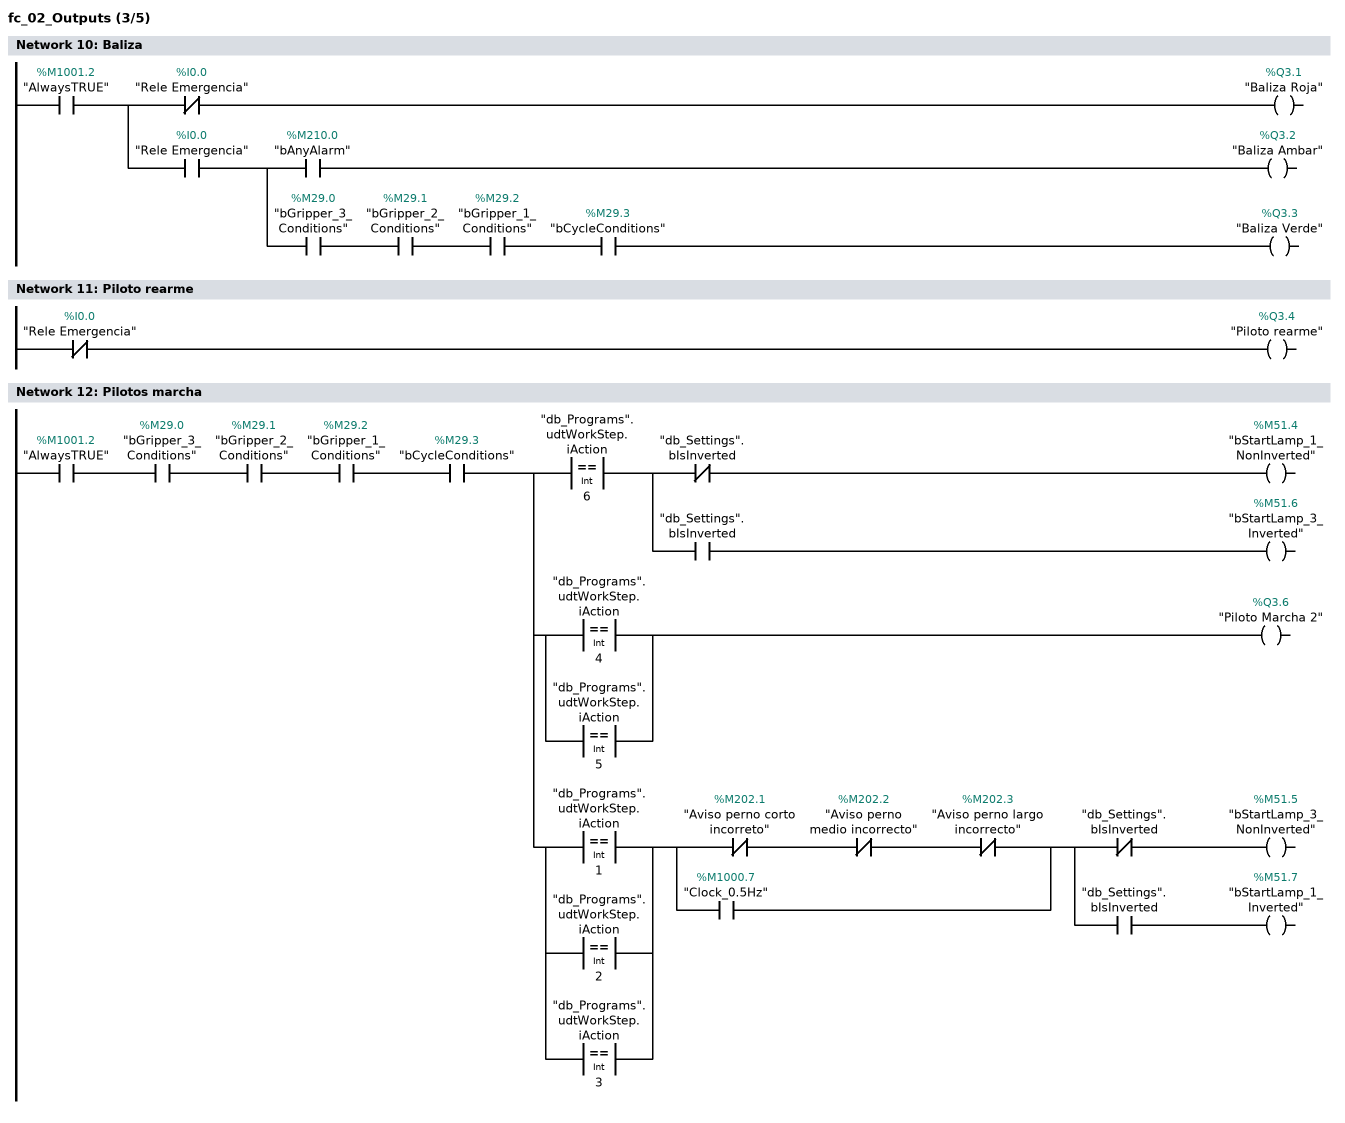
   RUNG wire#powerrail
      Contact( "AlwaysTRUE" )
      wire#w1
      I_Contact( "Rele Emergencia" )
      Coil( "Baliza Roja" )
   END_RUNG
   RUNG wire#w1
      Contact( "Rele Emergencia" )
      wire#w2
      Contact( "bAnyAlarm" )
      Coil( "Baliza Ambar" )
   END_RUNG
   RUNG wire#w2
      Contact( "bGripper_3_Conditions" )
      Contact( "bGripper_2_Conditions" )
      Contact( "bGripper_1_Conditions" )
      Contact( "bCycleConditions" )
      Coil( "Baliza Verde" )
   END_RUNG
   // the same network as SCL:
   "Baliza Roja" := "AlwaysTRUE" AND NOT "Rele Emergencia";
   #_w1 := "AlwaysTRUE" AND "Rele Emergencia";
   "Baliza Ambar" := #_w1 AND "bAnyAlarm";
   "Baliza Verde" := #_w1 AND "bGripper_3_Conditions" AND "bGripper_2_Conditions" AND "bGripper_1_Conditions" AND "bCycleConditions";
END_REGION

REGION Network 11: Piloto rearme
   RUNG wire#powerrail
      I_Contact( "Rele Emergencia" )
      Coil( "Piloto rearme" )
   END_RUNG
   // the same network as SCL:
   "Piloto rearme" := NOT "Rele Emergencia";
END_REGION

REGION Network 12: Pilotos marcha
   RUNG wire#powerrail
      Contact( "AlwaysTRUE" )
      Contact( "bGripper_3_Conditions" )
      Contact( "bGripper_2_Conditions" )
      Contact( "bGripper_1_Conditions" )
      Contact( "bCycleConditions" )
      wire#w1
      { S7_Templates := "SrcType := Int" } EQ_Contact(in1 := "db_Programs".udtWorkStep.iAction, in2 := 6)
      wire#w2
      I_Contact( "db_Settings".bIsInverted )
      Coil( "bStartLamp_1_NonInverted" )
   END_RUNG
   RUNG wire#w2
      Contact( "db_Settings".bIsInverted )
      Coil( "bStartLamp_3_Inverted" )
   END_RUNG
   RUNG wire#w1
      { S7_Templates := "SrcType := Int" } EQ_Contact(in1 := "db_Programs".udtWorkStep.iAction, in2 := 4)
      wire#w3
      Coil( "Piloto Marcha 2" )
   END_RUNG
   RUNG wire#w1
      { S7_Templates := "SrcType := Int" } EQ_Contact(in1 := "db_Programs".udtWorkStep.iAction, in2 := 5)
   END_RUNG wire#w3
   RUNG wire#w1
      { S7_Templates := "SrcType := Int" } EQ_Contact(in1 := "db_Programs".udtWorkStep.iAction, in2 := 1)
      wire#w4
      I_Contact( "Aviso perno corto incorreto" )
      I_Contact( "Aviso perno medio incorrecto" )
      I_Contact( "Aviso perno largo incorrecto" )
      wire#w5
      I_Contact( "db_Settings".bIsInverted )
      Coil( "bStartLamp_3_NonInverted" )
   END_RUNG
   RUNG wire#w1
      { S7_Templates := "SrcType := Int" } EQ_Contact(in1 := "db_Programs".udtWorkStep.iAction, in2 := 2)
   END_RUNG wire#w4
   RUNG wire#w1
      { S7_Templates := "SrcType := Int" } EQ_Contact(in1 := "db_Programs".udtWorkStep.iAction, in2 := 3)
   END_RUNG wire#w4
   RUNG wire#w4
      Contact( "Clock_0.5Hz" )
   END_RUNG wire#w5
   RUNG wire#w5
      Contact( "db_Settings".bIsInverted )
      Coil( "bStartLamp_1_Inverted" )
   END_RUNG
   // the same network as SCL:
   #_w1 := "AlwaysTRUE" AND "bGripper_3_Conditions" AND "bGripper_2_Conditions" AND "bGripper_1_Conditions" AND "bCycleConditions";
   #_w2 := #_w1 AND ("db_Programs".udtWorkStep.iAction = 6);
   "bStartLamp_1_NonInverted" := #_w2 AND NOT "db_Settings".bIsInverted;
   "bStartLamp_3_Inverted" := #_w2 AND "db_Settings".bIsInverted;
   "Piloto Marcha 2" := #_w1 AND (("db_Programs".udtWorkStep.iAction = 4) OR ("db_Programs".udtWorkStep.iAction = 5));
   #_w3 := #_w1 AND (("db_Programs".udtWorkStep.iAction = 1) OR ("db_Programs".udtWorkStep.iAction = 2) OR ("db_Programs".udtWorkStep.iAction = 3)) AND ((NOT "Aviso perno corto incorreto" AND NOT "Aviso perno medio incorrecto" AND NOT "Aviso perno largo incorrecto") OR "Clock_0.5Hz");
   "bStartLamp_3_NonInverted" := #_w3 AND NOT "db_Settings".bIsInverted;
   "bStartLamp_1_Inverted" := #_w3 AND "db_Settings".bIsInverted;
END_REGION

REGION Network 13: Pinzas
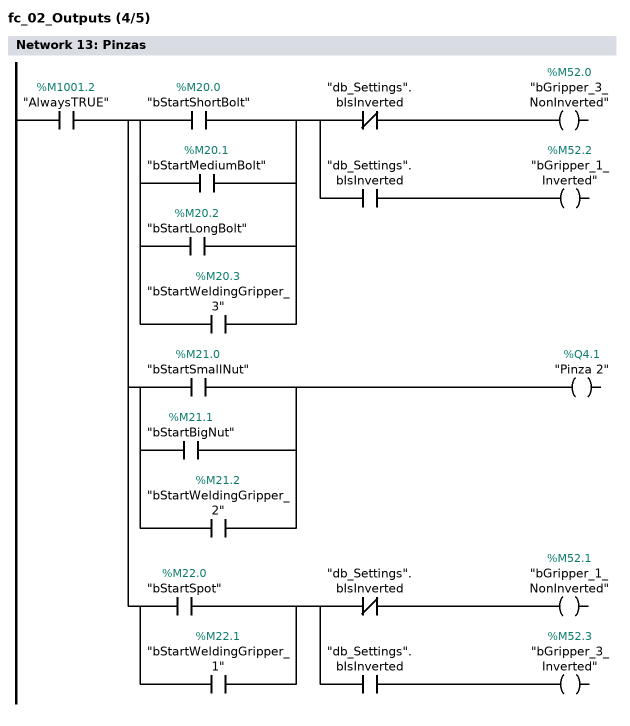
   RUNG wire#powerrail
      Contact( "AlwaysTRUE" )
      wire#w1
      Contact( "bStartShortBolt" )
      wire#w2
      I_Contact( "db_Settings".bIsInverted )
      Coil( "bGripper_3_NonInverted" )
   END_RUNG
   RUNG wire#w1
      Contact( "bStartMediumBolt" )
   END_RUNG wire#w2
   RUNG wire#w1
      Contact( "bStartLongBolt" )
   END_RUNG wire#w2
   RUNG wire#w1
      Contact( "bStartWeldingGripper_3" )
   END_RUNG wire#w2
   RUNG wire#w2
      Contact( "db_Settings".bIsInverted )
      Coil( "bGripper_1_Inverted" )
   END_RUNG
   RUNG wire#w1
      Contact( "bStartSmallNut" )
      wire#w3
      Coil( "Pinza 2" )
   END_RUNG
   RUNG wire#w1
      Contact( "bStartBigNut" )
   END_RUNG wire#w3
   RUNG wire#w1
      Contact( "bStartWeldingGripper_2" )
   END_RUNG wire#w3
   RUNG wire#w1
      Contact( "bStartSpot" )
      wire#w4
      I_Contact( "db_Settings".bIsInverted )
      Coil( "bGripper_1_NonInverted" )
   END_RUNG
   RUNG wire#w1
      Contact( "bStartWeldingGripper_1" )
   END_RUNG wire#w4
   RUNG wire#w4
      Contact( "db_Settings".bIsInverted )
      Coil( "bGripper_3_Inverted" )
   END_RUNG
   // the same network as SCL:
   #_w1 := "AlwaysTRUE" AND ("bStartShortBolt" OR "bStartMediumBolt" OR "bStartLongBolt" OR "bStartWeldingGripper_3");
   "bGripper_3_NonInverted" := #_w1 AND NOT "db_Settings".bIsInverted;
   "bGripper_1_Inverted" := #_w1 AND "db_Settings".bIsInverted;
   "Pinza 2" := "AlwaysTRUE" AND ("bStartSmallNut" OR "bStartBigNut" OR "bStartWeldingGripper_2");
   #_w2 := "AlwaysTRUE" AND ("bStartSpot" OR "bStartWeldingGripper_1");
   "bGripper_1_NonInverted" := #_w2 AND NOT "db_Settings".bIsInverted;
   "bGripper_3_Inverted" := #_w2 AND "db_Settings".bIsInverted;
END_REGION

REGION Network 14: Activación Salidas lámparas
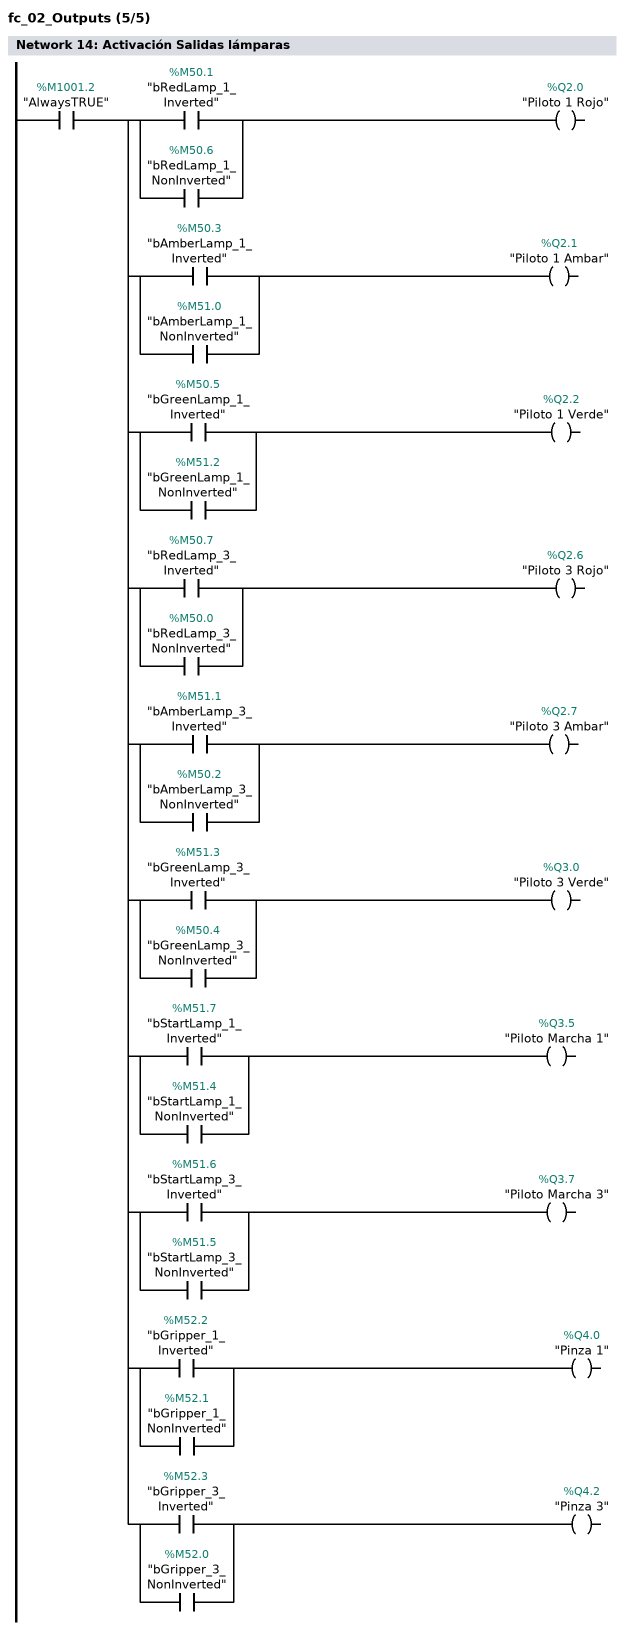
   RUNG wire#powerrail
      Contact( "AlwaysTRUE" )
      wire#w1
      Contact( "bRedLamp_1_Inverted" )
      wire#w2
      Coil( "Piloto 1 Rojo" )
   END_RUNG
   RUNG wire#w1
      Contact( "bRedLamp_1_NonInverted" )
   END_RUNG wire#w2
   RUNG wire#w1
      Contact( "bAmberLamp_1_Inverted" )
      wire#w3
      Coil( "Piloto 1 Ambar" )
   END_RUNG
   RUNG wire#w1
      Contact( "bAmberLamp_1_NonInverted" )
   END_RUNG wire#w3
   RUNG wire#w1
      Contact( "bGreenLamp_1_Inverted" )
      wire#w4
      Coil( "Piloto 1 Verde" )
   END_RUNG
   RUNG wire#w1
      Contact( "bGreenLamp_1_NonInverted" )
   END_RUNG wire#w4
   RUNG wire#w1
      Contact( "bRedLamp_3_Inverted" )
      wire#w5
      Coil( "Piloto 3 Rojo" )
   END_RUNG
   RUNG wire#w1
      Contact( "bRedLamp_3_NonInverted" )
   END_RUNG wire#w5
   RUNG wire#w1
      Contact( "bAmberLamp_3_Inverted" )
      wire#w6
      Coil( "Piloto 3 Ambar" )
   END_RUNG
   RUNG wire#w1
      Contact( "bAmberLamp_3_NonInverted" )
   END_RUNG wire#w6
   RUNG wire#w1
      Contact( "bGreenLamp_3_Inverted" )
      wire#w7
      Coil( "Piloto 3 Verde" )
   END_RUNG
   RUNG wire#w1
      Contact( "bGreenLamp_3_NonInverted" )
   END_RUNG wire#w7
   RUNG wire#w1
      Contact( "bStartLamp_1_Inverted" )
      wire#w8
      Coil( "Piloto Marcha 1" )
   END_RUNG
   RUNG wire#w1
      Contact( "bStartLamp_1_NonInverted" )
   END_RUNG wire#w8
   RUNG wire#w1
      Contact( "bStartLamp_3_Inverted" )
      wire#w9
      Coil( "Piloto Marcha 3" )
   END_RUNG
   RUNG wire#w1
      Contact( "bStartLamp_3_NonInverted" )
   END_RUNG wire#w9
   RUNG wire#w1
      Contact( "bGripper_1_Inverted" )
      wire#w10
      Coil( "Pinza 1" )
   END_RUNG
   RUNG wire#w1
      Contact( "bGripper_1_NonInverted" )
   END_RUNG wire#w10
   RUNG wire#w1
      Contact( "bGripper_3_Inverted" )
      wire#w11
      Coil( "Pinza 3" )
   END_RUNG
   RUNG wire#w1
      Contact( "bGripper_3_NonInverted" )
   END_RUNG wire#w11
   // the same network as SCL:
   "Piloto 1 Rojo" := "AlwaysTRUE" AND ("bRedLamp_1_Inverted" OR "bRedLamp_1_NonInverted");
   "Piloto 1 Ambar" := "AlwaysTRUE" AND ("bAmberLamp_1_Inverted" OR "bAmberLamp_1_NonInverted");
   "Piloto 1 Verde" := "AlwaysTRUE" AND ("bGreenLamp_1_Inverted" OR "bGreenLamp_1_NonInverted");
   "Piloto 3 Rojo" := "AlwaysTRUE" AND ("bRedLamp_3_Inverted" OR "bRedLamp_3_NonInverted");
   "Piloto 3 Ambar" := "AlwaysTRUE" AND ("bAmberLamp_3_Inverted" OR "bAmberLamp_3_NonInverted");
   "Piloto 3 Verde" := "AlwaysTRUE" AND ("bGreenLamp_3_Inverted" OR "bGreenLamp_3_NonInverted");
   "Piloto Marcha 1" := "AlwaysTRUE" AND ("bStartLamp_1_Inverted" OR "bStartLamp_1_NonInverted");
   "Piloto Marcha 3" := "AlwaysTRUE" AND ("bStartLamp_3_Inverted" OR "bStartLamp_3_NonInverted");
   "Pinza 1" := "AlwaysTRUE" AND ("bGripper_1_Inverted" OR "bGripper_1_NonInverted");
   "Pinza 3" := "AlwaysTRUE" AND ("bGripper_3_Inverted" OR "bGripper_3_NonInverted");
END_REGION
END_FUNCTION

FUNCTION "fc_03_Alarms" : Void   // FC3, LAD
{ S7_Optimized_Access := 'TRUE' }
VERSION : 0.1
// stored: AutoNumber false, IsIECCheckEnabled false, SetENOAutomatically false, UDAEnableTagReadback false
   VAR_TEMP   // added for the SCL form of the ladder/FBD networks
      _w1 : Bool;
      _w2 : Bool;
      _w3 : Bool;
   END_VAR
BEGIN

REGION Network 1
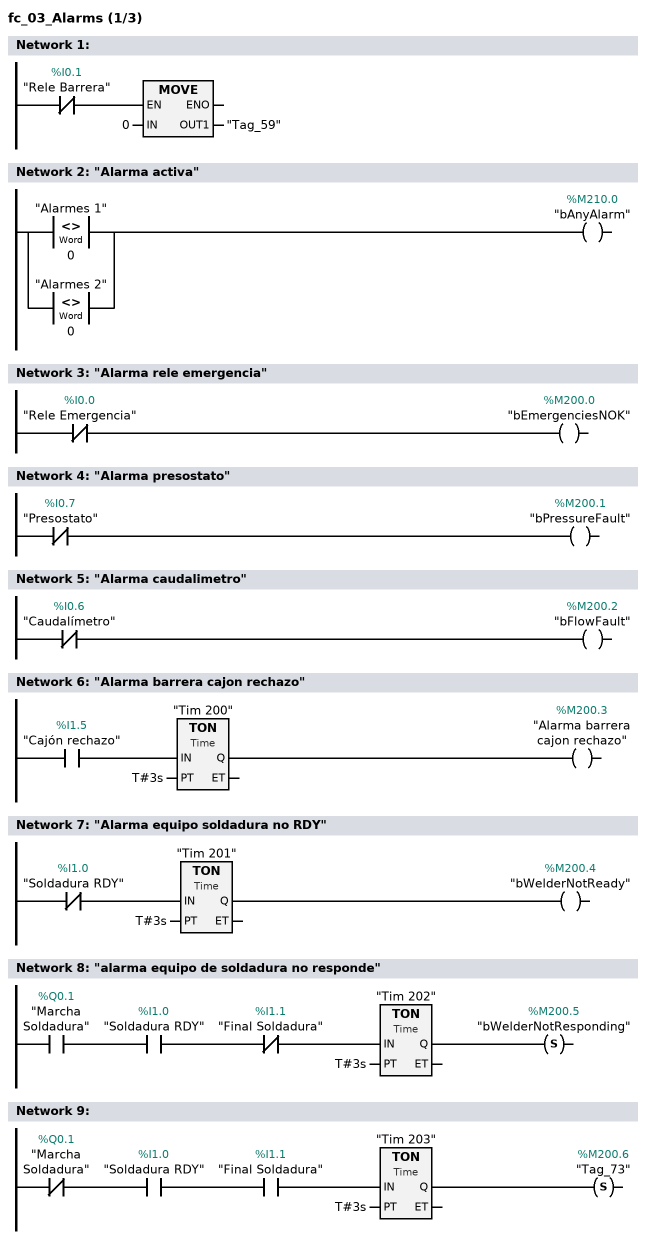
   RUNG wire#powerrail
      I_Contact( "Rele Barrera" )
      Move(in := 0, out1 => "Tag_59")
   END_RUNG
   // the same network as SCL:
   IF NOT "Rele Barrera" THEN "Tag_59" := 0; END_IF;
END_REGION

REGION Network 2: "Alarma activa"
   RUNG wire#powerrail
      { S7_Templates := "SrcType := Word" } NE_Contact(in1 := "Alarmes 1", in2 := 0)
      wire#w1
      Coil( "bAnyAlarm" )
   END_RUNG
   RUNG wire#powerrail
      { S7_Templates := "SrcType := Word" } NE_Contact(in1 := "Alarmes 2", in2 := 0)
   END_RUNG wire#w1
   // the same network as SCL:
   "bAnyAlarm" := ("Alarmes 1" <> 0) OR ("Alarmes 2" <> 0);
END_REGION

REGION Network 3: "Alarma rele emergencia"
   RUNG wire#powerrail
      I_Contact( "Rele Emergencia" )
      Coil( "bEmergenciesNOK" )
   END_RUNG
   // the same network as SCL:
   "bEmergenciesNOK" := NOT "Rele Emergencia";
END_REGION

REGION Network 4: "Alarma presostato"
   RUNG wire#powerrail
      I_Contact( "Presostato" )
      Coil( "bPressureFault" )
   END_RUNG
   // the same network as SCL:
   "bPressureFault" := NOT "Presostato";
END_REGION

REGION Network 5: "Alarma caudalimetro"
   RUNG wire#powerrail
      I_Contact( "Caudalímetro" )
      Coil( "bFlowFault" )
   END_RUNG
   // the same network as SCL:
   "bFlowFault" := NOT "Caudalímetro";
END_REGION

REGION Network 6: "Alarma barrera cajon rechazo"
   RUNG wire#powerrail
      Contact( "Cajón rechazo" )
      { S7_Templates := "time_type := Time" } "Tim 200".TON(pt := T#3s, et =>)
      Coil( "Alarma barrera cajon rechazo" )
   END_RUNG
   // the same network as SCL:
   "Tim 200".TON(IN := "Cajón rechazo", PT := T#3s);
   "Alarma barrera cajon rechazo" := "Tim 200".Q;
END_REGION

REGION Network 7: "Alarma equipo soldadura no RDY"
   RUNG wire#powerrail
      I_Contact( "Soldadura RDY" )
      { S7_Templates := "time_type := Time" } "Tim 201".TON(pt := T#3s, et =>)
      Coil( "bWelderNotReady" )
   END_RUNG
   // the same network as SCL:
   "Tim 201".TON(IN := NOT "Soldadura RDY", PT := T#3s);
   "bWelderNotReady" := "Tim 201".Q;
END_REGION

REGION Network 8: "alarma equipo de soldadura no responde"
   RUNG wire#powerrail
      Contact( "Marcha Soldadura" )
      Contact( "Soldadura RDY" )
      I_Contact( "Final Soldadura" )
      { S7_Templates := "time_type := Time" } "Tim 202".TON(pt := T#3s, et =>)
      S_Coil( "bWelderNotResponding" )
   END_RUNG
   // the same network as SCL:
   "Tim 202".TON(IN := "Marcha Soldadura" AND "Soldadura RDY" AND NOT "Final Soldadura", PT := T#3s);
   IF "Tim 202".Q THEN "bWelderNotResponding" := TRUE; END_IF;
END_REGION

REGION Network 9
   RUNG wire#powerrail
      I_Contact( "Marcha Soldadura" )
      Contact( "Soldadura RDY" )
      Contact( "Final Soldadura" )
      { S7_Templates := "time_type := Time" } "Tim 203".TON(pt := T#3s, et =>)
      S_Coil( "Tag_73" )
   END_RUNG
   // the same network as SCL:
   "Tim 203".TON(IN := NOT "Marcha Soldadura" AND "Soldadura RDY" AND "Final Soldadura", PT := T#3s);
   IF "Tim 203".Q THEN "Tag_73" := TRUE; END_IF;
END_REGION

REGION Network 10
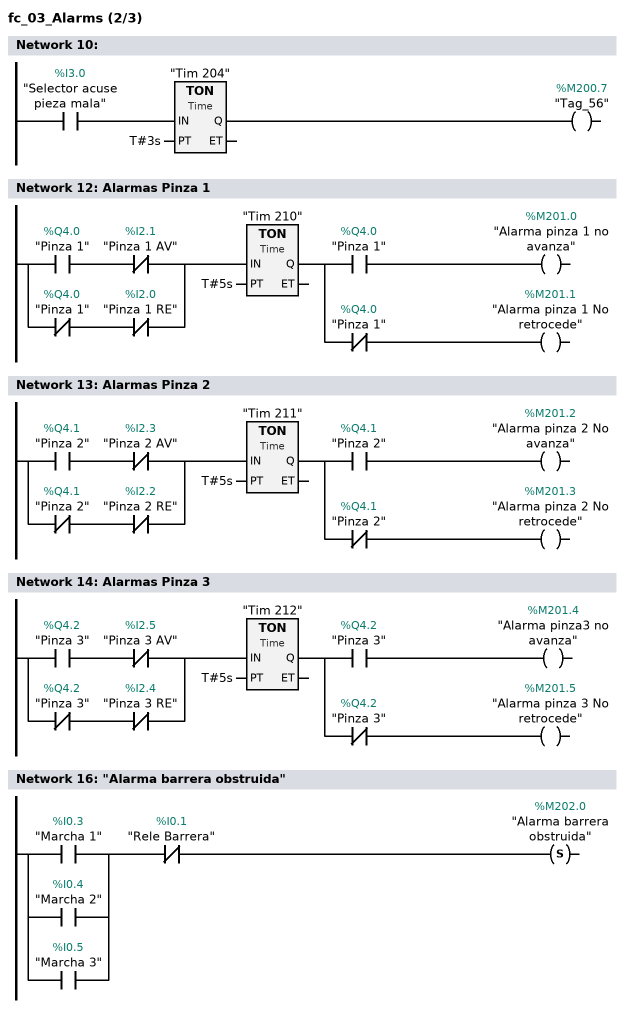
   RUNG wire#powerrail
      Contact( "Selector acuse pieza mala" )
      { S7_Templates := "time_type := Time" } "Tim 204".TON(pt := T#3s, et =>)
      Coil( "Tag_56" )
   END_RUNG
   // the same network as SCL:
   "Tim 204".TON(IN := "Selector acuse pieza mala", PT := T#3s);
   "Tag_56" := "Tim 204".Q;
END_REGION

REGION Network 12: Alarmas Pinza 1
   RUNG wire#powerrail
      Contact( "Pinza 1" )
      I_Contact( "Pinza 1 AV" )
      wire#w1
      { S7_Templates := "time_type := Time" } "Tim 210".TON(pt := T#5s, et =>)
      wire#w2
      Contact( "Pinza 1" )
      Coil( "Alarma pinza 1 no avanza" )
   END_RUNG
   RUNG wire#powerrail
      I_Contact( "Pinza 1" )
      I_Contact( "Pinza 1 RE" )
   END_RUNG wire#w1
   RUNG wire#w2
      I_Contact( "Pinza 1" )
      Coil( "Alarma pinza 1 No retrocede" )
   END_RUNG
   // the same network as SCL:
   "Tim 210".TON(IN := ("Pinza 1" AND NOT "Pinza 1 AV") OR (NOT "Pinza 1" AND NOT "Pinza 1 RE"), PT := T#5s);
   "Alarma pinza 1 no avanza" := "Tim 210".Q AND "Pinza 1";
   "Alarma pinza 1 No retrocede" := "Tim 210".Q AND NOT "Pinza 1";
END_REGION

REGION Network 13: Alarmas Pinza 2
   RUNG wire#powerrail
      Contact( "Pinza 2" )
      I_Contact( "Pinza 2 AV" )
      wire#w1
      { S7_Templates := "time_type := Time" } "Tim 211".TON(pt := T#5s, et =>)
      wire#w2
      Contact( "Pinza 2" )
      Coil( "Alarma pinza 2 No avanza" )
   END_RUNG
   RUNG wire#powerrail
      I_Contact( "Pinza 2" )
      I_Contact( "Pinza 2 RE" )
   END_RUNG wire#w1
   RUNG wire#w2
      I_Contact( "Pinza 2" )
      Coil( "Alarma pinza 2 No retrocede" )
   END_RUNG
   // the same network as SCL:
   "Tim 211".TON(IN := ("Pinza 2" AND NOT "Pinza 2 AV") OR (NOT "Pinza 2" AND NOT "Pinza 2 RE"), PT := T#5s);
   "Alarma pinza 2 No avanza" := "Tim 211".Q AND "Pinza 2";
   "Alarma pinza 2 No retrocede" := "Tim 211".Q AND NOT "Pinza 2";
END_REGION

REGION Network 14: Alarmas Pinza 3
   RUNG wire#powerrail
      Contact( "Pinza 3" )
      I_Contact( "Pinza 3 AV" )
      wire#w1
      { S7_Templates := "time_type := Time" } "Tim 212".TON(pt := T#5s, et =>)
      wire#w2
      Contact( "Pinza 3" )
      Coil( "Alarma pinza3 no avanza" )
   END_RUNG
   RUNG wire#powerrail
      I_Contact( "Pinza 3" )
      I_Contact( "Pinza 3 RE" )
   END_RUNG wire#w1
   RUNG wire#w2
      I_Contact( "Pinza 3" )
      Coil( "Alarma pinza 3 No retrocede" )
   END_RUNG
   // the same network as SCL:
   "Tim 212".TON(IN := ("Pinza 3" AND NOT "Pinza 3 AV") OR (NOT "Pinza 3" AND NOT "Pinza 3 RE"), PT := T#5s);
   "Alarma pinza3 no avanza" := "Tim 212".Q AND "Pinza 3";
   "Alarma pinza 3 No retrocede" := "Tim 212".Q AND NOT "Pinza 3";
END_REGION

REGION Network 16: "Alarma barrera obstruida"
   RUNG wire#powerrail
      Contact( "Marcha 1" )
      wire#w1
      I_Contact( "Rele Barrera" )
      S_Coil( "Alarma barrera obstruida" )
   END_RUNG
   RUNG wire#powerrail
      Contact( "Marcha 2" )
   END_RUNG wire#w1
   RUNG wire#powerrail
      Contact( "Marcha 3" )
   END_RUNG wire#w1
   // the same network as SCL:
   IF ("Marcha 1" OR "Marcha 2" OR "Marcha 3") AND NOT "Rele Barrera" THEN
       "Alarma barrera obstruida" := TRUE;
   END_IF;
END_REGION

REGION Network 17: Avisos perno incorrecto
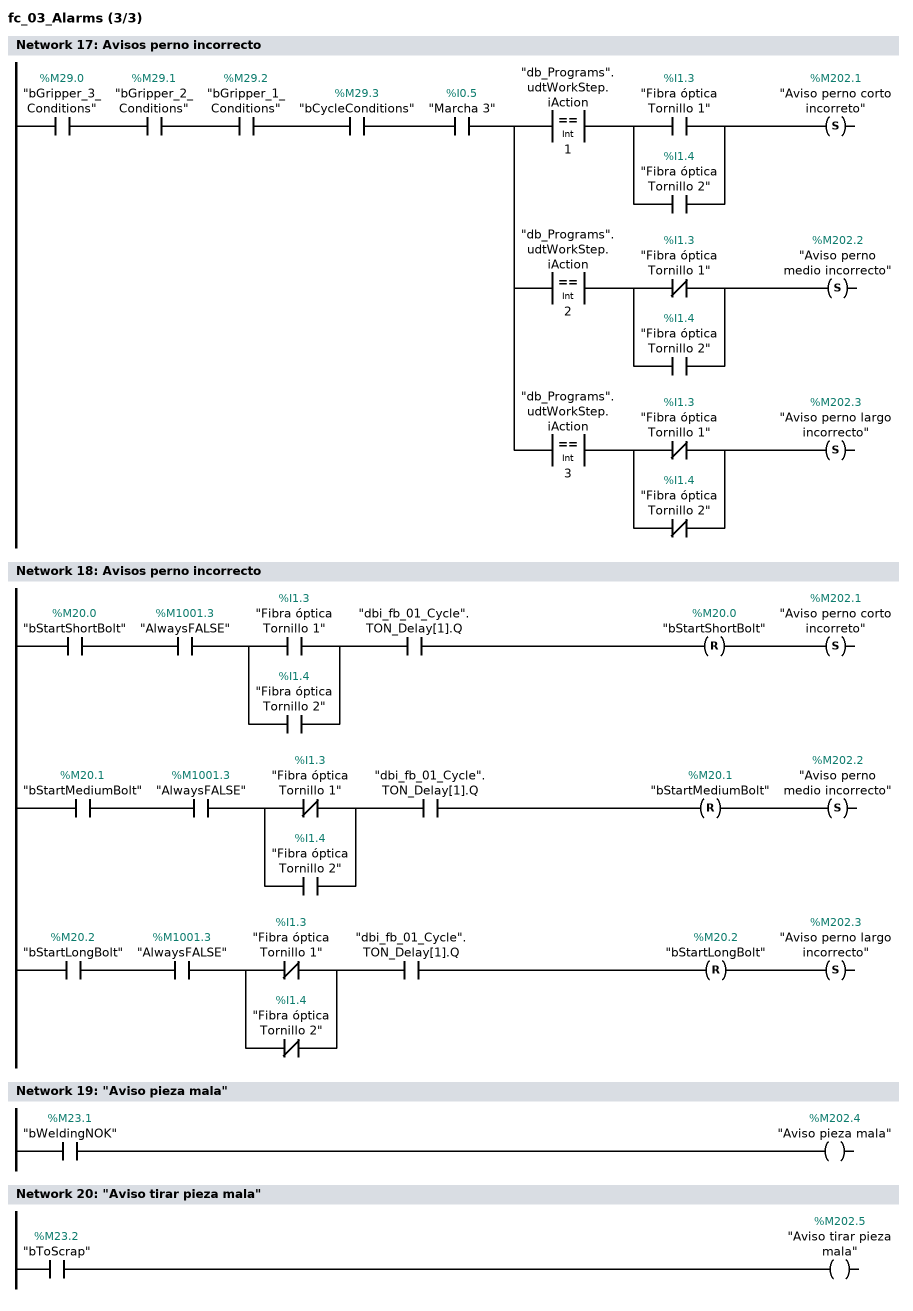
   RUNG wire#powerrail
      Contact( "bGripper_3_Conditions" )
      Contact( "bGripper_2_Conditions" )
      Contact( "bGripper_1_Conditions" )
      Contact( "bCycleConditions" )
      Contact( "Marcha 3" )
      wire#w1
      { S7_Templates := "SrcType := Int" } EQ_Contact(in1 := "db_Programs".udtWorkStep.iAction, in2 := 1)
      wire#w2
      Contact( "Fibra óptica Tornillo 1" )
      wire#w3
      S_Coil( "Aviso perno corto incorreto" )
   END_RUNG
   RUNG wire#w2
      Contact( "Fibra óptica Tornillo 2" )
   END_RUNG wire#w3
   RUNG wire#w1
      { S7_Templates := "SrcType := Int" } EQ_Contact(in1 := "db_Programs".udtWorkStep.iAction, in2 := 2)
      wire#w4
      I_Contact( "Fibra óptica Tornillo 1" )
      wire#w5
      S_Coil( "Aviso perno medio incorrecto" )
   END_RUNG
   RUNG wire#w4
      Contact( "Fibra óptica Tornillo 2" )
   END_RUNG wire#w5
   RUNG wire#w1
      { S7_Templates := "SrcType := Int" } EQ_Contact(in1 := "db_Programs".udtWorkStep.iAction, in2 := 3)
      wire#w6
      I_Contact( "Fibra óptica Tornillo 1" )
      wire#w7
      S_Coil( "Aviso perno largo incorrecto" )
   END_RUNG
   RUNG wire#w6
      I_Contact( "Fibra óptica Tornillo 2" )
   END_RUNG wire#w7
   // the same network as SCL:
   #_w1 := "bGripper_3_Conditions" AND "bGripper_2_Conditions" AND "bGripper_1_Conditions" AND "bCycleConditions" AND "Marcha 3";
   IF #_w1 AND ("db_Programs".udtWorkStep.iAction = 1) AND ("Fibra óptica Tornillo 1" OR "Fibra óptica Tornillo 2") THEN
       "Aviso perno corto incorreto" := TRUE;
   END_IF;
   IF #_w1 AND ("db_Programs".udtWorkStep.iAction = 2) AND (NOT "Fibra óptica Tornillo 1" OR "Fibra óptica Tornillo 2") THEN
       "Aviso perno medio incorrecto" := TRUE;
   END_IF;
   IF #_w1 AND ("db_Programs".udtWorkStep.iAction = 3) AND (NOT "Fibra óptica Tornillo 1" OR NOT "Fibra óptica Tornillo 2") THEN
       "Aviso perno largo incorrecto" := TRUE;
   END_IF;
END_REGION

REGION Network 18: Avisos perno incorrecto
   RUNG wire#powerrail
      Contact( "bStartShortBolt" )
      Contact( "AlwaysFALSE" )
      wire#w1
      Contact( "Fibra óptica Tornillo 1" )
      wire#w2
      Contact( "dbi_fb_01_Cycle".TON_Delay[1].Q )
      R_Coil( "bStartShortBolt" )
      S_Coil( "Aviso perno corto incorreto" )
   END_RUNG
   RUNG wire#w1
      Contact( "Fibra óptica Tornillo 2" )
   END_RUNG wire#w2
   RUNG wire#powerrail
      Contact( "bStartMediumBolt" )
      Contact( "AlwaysFALSE" )
      wire#w3
      I_Contact( "Fibra óptica Tornillo 1" )
      wire#w4
      Contact( "dbi_fb_01_Cycle".TON_Delay[1].Q )
      R_Coil( "bStartMediumBolt" )
      S_Coil( "Aviso perno medio incorrecto" )
   END_RUNG
   RUNG wire#w3
      Contact( "Fibra óptica Tornillo 2" )
   END_RUNG wire#w4
   RUNG wire#powerrail
      Contact( "bStartLongBolt" )
      Contact( "AlwaysFALSE" )
      wire#w5
      I_Contact( "Fibra óptica Tornillo 1" )
      wire#w6
      Contact( "dbi_fb_01_Cycle".TON_Delay[1].Q )
      R_Coil( "bStartLongBolt" )
      S_Coil( "Aviso perno largo incorrecto" )
   END_RUNG
   RUNG wire#w5
      I_Contact( "Fibra óptica Tornillo 2" )
   END_RUNG wire#w6
   // the same network as SCL:
   #_w1 := "bStartShortBolt" AND "AlwaysFALSE" AND ("Fibra óptica Tornillo 1" OR "Fibra óptica Tornillo 2") AND "dbi_fb_01_Cycle".TON_Delay[1].Q;
   IF #_w1 THEN
       "bStartShortBolt" := FALSE;
       "Aviso perno corto incorreto" := TRUE;
   END_IF;
   #_w2 := "bStartMediumBolt" AND "AlwaysFALSE" AND (NOT "Fibra óptica Tornillo 1" OR "Fibra óptica Tornillo 2") AND "dbi_fb_01_Cycle".TON_Delay[1].Q;
   IF #_w2 THEN
       "bStartMediumBolt" := FALSE;
       "Aviso perno medio incorrecto" := TRUE;
   END_IF;
   #_w3 := "bStartLongBolt" AND "AlwaysFALSE" AND (NOT "Fibra óptica Tornillo 1" OR NOT "Fibra óptica Tornillo 2") AND "dbi_fb_01_Cycle".TON_Delay[1].Q;
   IF #_w3 THEN
       "bStartLongBolt" := FALSE;
       "Aviso perno largo incorrecto" := TRUE;
   END_IF;
END_REGION

REGION Network 19: "Aviso pieza mala"
   RUNG wire#powerrail
      Contact( "bWeldingNOK" )
      Coil( "Aviso pieza mala" )
   END_RUNG
   // the same network as SCL:
   "Aviso pieza mala" := "bWeldingNOK";
END_REGION

REGION Network 20: "Aviso tirar pieza mala"
   RUNG wire#powerrail
      Contact( "bToScrap" )
      Coil( "Aviso tirar pieza mala" )
   END_RUNG
   // the same network as SCL:
   "Aviso tirar pieza mala" := "bToScrap";
END_REGION
END_FUNCTION

FUNCTION "fc_04_HMI" : Void   // FC4, LAD
{ S7_Optimized_Access := 'TRUE' }
VERSION : 0.1
// stored: AutoNumber false, IsIECCheckEnabled false, SetENOAutomatically false, UDAEnableTagReadback false
   VAR_TEMP   // added for the SCL form of the ladder/FBD networks
      _w1 : Bool;
      _w2 : Bool;
      _w3 : Bool;
   END_VAR
BEGIN

REGION Network 1
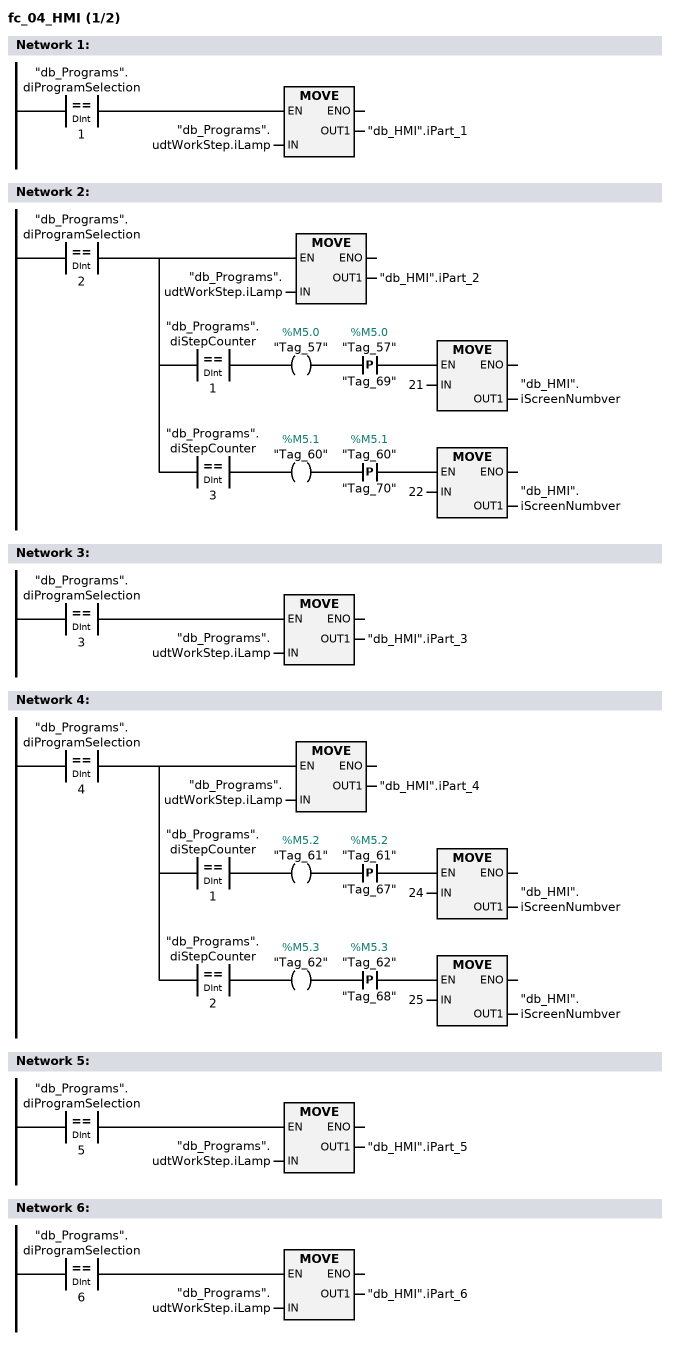
   RUNG wire#powerrail
      { S7_Templates := "SrcType := DInt" } EQ_Contact(in1 := "db_Programs".diProgramSelection, in2 := 1)
      Move(in := "db_Programs".udtWorkStep.iLamp, out1 => "db_HMI".iPart_1)
   END_RUNG
   // the same network as SCL:
   IF "db_Programs".diProgramSelection = 1 THEN "db_HMI".iPart_1 := "db_Programs".udtWorkStep.iLamp; END_IF;
END_REGION

REGION Network 2
   RUNG wire#powerrail
      { S7_Templates := "SrcType := DInt" } EQ_Contact(in1 := "db_Programs".diProgramSelection, in2 := 2)
      wire#w1
      Move(in := "db_Programs".udtWorkStep.iLamp, out1 => "db_HMI".iPart_2)
   END_RUNG
   RUNG wire#w1
      { S7_Templates := "SrcType := DInt" } EQ_Contact(in1 := "db_Programs".diStepCounter, in2 := 1)
      Coil( "Tag_57" )
      P_Contact(operand := "Tag_57", bit := "Tag_69")
      Move(in := 21, out1 => "db_HMI".iScreenNumbver)
   END_RUNG
   RUNG wire#w1
      { S7_Templates := "SrcType := DInt" } EQ_Contact(in1 := "db_Programs".diStepCounter, in2 := 3)
      Coil( "Tag_60" )
      P_Contact(operand := "Tag_60", bit := "Tag_70")
      Move(in := 22, out1 => "db_HMI".iScreenNumbver)
   END_RUNG
   // the same network as SCL:
   #_w1 := "db_Programs".diProgramSelection = 2;
   IF #_w1 THEN "db_HMI".iPart_2 := "db_Programs".udtWorkStep.iLamp; END_IF;
   "Tag_57" := #_w1 AND ("db_Programs".diStepCounter = 1);
   #_w2 := "Tag_57" AND "Tag_57" AND NOT "Tag_69";   // rising edge of "Tag_57"
   "Tag_69" := "Tag_57";
   IF #_w2 THEN "db_HMI".iScreenNumbver := 21; END_IF;
   "Tag_60" := #_w1 AND ("db_Programs".diStepCounter = 3);
   #_w3 := "Tag_60" AND "Tag_60" AND NOT "Tag_70";   // rising edge of "Tag_60"
   "Tag_70" := "Tag_60";
   IF #_w3 THEN "db_HMI".iScreenNumbver := 22; END_IF;
END_REGION

REGION Network 3
   RUNG wire#powerrail
      { S7_Templates := "SrcType := DInt" } EQ_Contact(in1 := "db_Programs".diProgramSelection, in2 := 3)
      Move(in := "db_Programs".udtWorkStep.iLamp, out1 => "db_HMI".iPart_3)
   END_RUNG
   // the same network as SCL:
   IF "db_Programs".diProgramSelection = 3 THEN "db_HMI".iPart_3 := "db_Programs".udtWorkStep.iLamp; END_IF;
END_REGION

REGION Network 4
   RUNG wire#powerrail
      { S7_Templates := "SrcType := DInt" } EQ_Contact(in1 := "db_Programs".diProgramSelection, in2 := 4)
      wire#w1
      Move(in := "db_Programs".udtWorkStep.iLamp, out1 => "db_HMI".iPart_4)
   END_RUNG
   RUNG wire#w1
      { S7_Templates := "SrcType := DInt" } EQ_Contact(in1 := "db_Programs".diStepCounter, in2 := 1)
      Coil( "Tag_61" )
      P_Contact(operand := "Tag_61", bit := "Tag_67")
      Move(in := 24, out1 => "db_HMI".iScreenNumbver)
   END_RUNG
   RUNG wire#w1
      { S7_Templates := "SrcType := DInt" } EQ_Contact(in1 := "db_Programs".diStepCounter, in2 := 2)
      Coil( "Tag_62" )
      P_Contact(operand := "Tag_62", bit := "Tag_68")
      Move(in := 25, out1 => "db_HMI".iScreenNumbver)
   END_RUNG
   // the same network as SCL:
   #_w1 := "db_Programs".diProgramSelection = 4;
   IF #_w1 THEN "db_HMI".iPart_4 := "db_Programs".udtWorkStep.iLamp; END_IF;
   "Tag_61" := #_w1 AND ("db_Programs".diStepCounter = 1);
   #_w2 := "Tag_61" AND "Tag_61" AND NOT "Tag_67";   // rising edge of "Tag_61"
   "Tag_67" := "Tag_61";
   IF #_w2 THEN "db_HMI".iScreenNumbver := 24; END_IF;
   "Tag_62" := #_w1 AND ("db_Programs".diStepCounter = 2);
   #_w3 := "Tag_62" AND "Tag_62" AND NOT "Tag_68";   // rising edge of "Tag_62"
   "Tag_68" := "Tag_62";
   IF #_w3 THEN "db_HMI".iScreenNumbver := 25; END_IF;
END_REGION

REGION Network 5
   RUNG wire#powerrail
      { S7_Templates := "SrcType := DInt" } EQ_Contact(in1 := "db_Programs".diProgramSelection, in2 := 5)
      Move(in := "db_Programs".udtWorkStep.iLamp, out1 => "db_HMI".iPart_5)
   END_RUNG
   // the same network as SCL:
   IF "db_Programs".diProgramSelection = 5 THEN "db_HMI".iPart_5 := "db_Programs".udtWorkStep.iLamp; END_IF;
END_REGION

REGION Network 6
   RUNG wire#powerrail
      { S7_Templates := "SrcType := DInt" } EQ_Contact(in1 := "db_Programs".diProgramSelection, in2 := 6)
      Move(in := "db_Programs".udtWorkStep.iLamp, out1 => "db_HMI".iPart_6)
   END_RUNG
   // the same network as SCL:
   IF "db_Programs".diProgramSelection = 6 THEN "db_HMI".iPart_6 := "db_Programs".udtWorkStep.iLamp; END_IF;
END_REGION

REGION Network 7
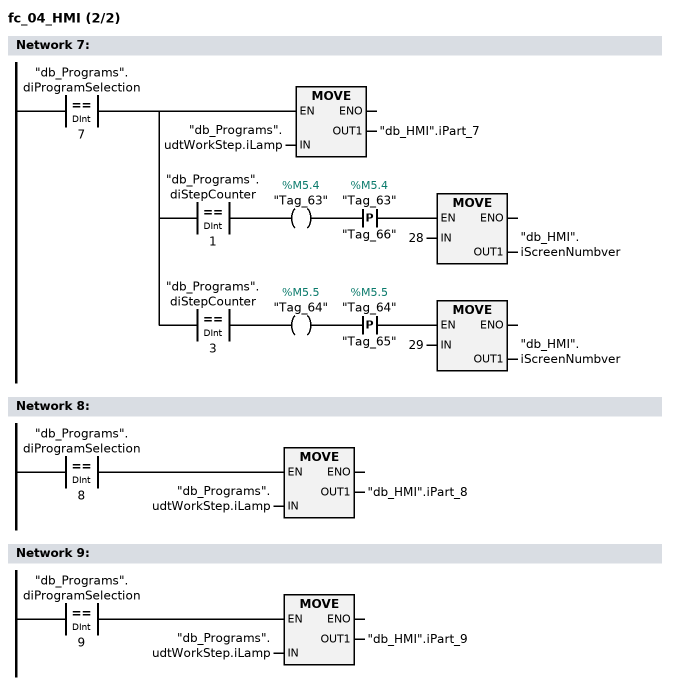
   RUNG wire#powerrail
      { S7_Templates := "SrcType := DInt" } EQ_Contact(in1 := "db_Programs".diProgramSelection, in2 := 7)
      wire#w1
      Move(in := "db_Programs".udtWorkStep.iLamp, out1 => "db_HMI".iPart_7)
   END_RUNG
   RUNG wire#w1
      { S7_Templates := "SrcType := DInt" } EQ_Contact(in1 := "db_Programs".diStepCounter, in2 := 1)
      Coil( "Tag_63" )
      P_Contact(operand := "Tag_63", bit := "Tag_66")
      Move(in := 28, out1 => "db_HMI".iScreenNumbver)
   END_RUNG
   RUNG wire#w1
      { S7_Templates := "SrcType := DInt" } EQ_Contact(in1 := "db_Programs".diStepCounter, in2 := 3)
      Coil( "Tag_64" )
      P_Contact(operand := "Tag_64", bit := "Tag_65")
      Move(in := 29, out1 => "db_HMI".iScreenNumbver)
   END_RUNG
   // the same network as SCL:
   #_w1 := "db_Programs".diProgramSelection = 7;
   IF #_w1 THEN "db_HMI".iPart_7 := "db_Programs".udtWorkStep.iLamp; END_IF;
   "Tag_63" := #_w1 AND ("db_Programs".diStepCounter = 1);
   #_w2 := "Tag_63" AND "Tag_63" AND NOT "Tag_66";   // rising edge of "Tag_63"
   "Tag_66" := "Tag_63";
   IF #_w2 THEN "db_HMI".iScreenNumbver := 28; END_IF;
   "Tag_64" := #_w1 AND ("db_Programs".diStepCounter = 3);
   #_w3 := "Tag_64" AND "Tag_64" AND NOT "Tag_65";   // rising edge of "Tag_64"
   "Tag_65" := "Tag_64";
   IF #_w3 THEN "db_HMI".iScreenNumbver := 29; END_IF;
END_REGION

REGION Network 8
   RUNG wire#powerrail
      { S7_Templates := "SrcType := DInt" } EQ_Contact(in1 := "db_Programs".diProgramSelection, in2 := 8)
      Move(in := "db_Programs".udtWorkStep.iLamp, out1 => "db_HMI".iPart_8)
   END_RUNG
   // the same network as SCL:
   IF "db_Programs".diProgramSelection = 8 THEN "db_HMI".iPart_8 := "db_Programs".udtWorkStep.iLamp; END_IF;
END_REGION

REGION Network 9
   RUNG wire#powerrail
      { S7_Templates := "SrcType := DInt" } EQ_Contact(in1 := "db_Programs".diProgramSelection, in2 := 9)
      Move(in := "db_Programs".udtWorkStep.iLamp, out1 => "db_HMI".iPart_9)
   END_RUNG
   // the same network as SCL:
   IF "db_Programs".diProgramSelection = 9 THEN "db_HMI".iPart_9 := "db_Programs".udtWorkStep.iLamp; END_IF;
END_REGION
END_FUNCTION

FUNCTION "fc_05_Analog" : Void   // FC5, LAD
{ S7_Optimized_Access := 'TRUE' }
VERSION : 0.1
// stored: AutoNumber true, IsIECCheckEnabled false, SetENOAutomatically false, UDAEnableTagReadback false
BEGIN

REGION Network 1
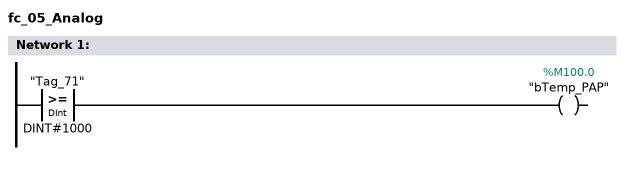
   RUNG wire#powerrail
      { S7_Templates := "SrcType := DInt" } GE_Contact(in1 := "Tag_71", in2 := DINT#1000)
      Coil( "bTemp_PAP" )
   END_RUNG
   // the same network as SCL:
   "bTemp_PAP" := "Tag_71" >= DINT#1000;
END_REGION
END_FUNCTION

DATA_BLOCK "dbi_fb_01_Cycle"   // DB1
VERSION : 0.1
// stored: AutoNumber false, InstanceOfName fb_01_Cycle, InstanceOfType FB
"fb_01_Cycle"
BEGIN
END_DATA_BLOCK

DATA_BLOCK "Tim 200"   // DB200
{ S7_Optimized_Access := 'TRUE' }
// stored: AutoNumber false, InstanceOfName IEC_TIMER, OfSystemLibElement IEC_TIMER, OfSystemLibVersion 1.0
"IEC_TIMER"
   // VAR
   //    PT : Time;
   //    ET { ExternalWritable := 'False'} : Time;
   //    IN : Bool;
   //    Q { ExternalWritable := 'False'} : Bool;
   // END_VAR
BEGIN
END_DATA_BLOCK

DATA_BLOCK "Tim 201"   // DB201
{ S7_Optimized_Access := 'TRUE' }
// stored: AutoNumber false, InstanceOfName IEC_TIMER, OfSystemLibElement IEC_TIMER, OfSystemLibVersion 1.0
"IEC_TIMER"
   // VAR
   //    PT : Time;
   //    ET { ExternalWritable := 'False'} : Time;
   //    IN : Bool;
   //    Q { ExternalWritable := 'False'} : Bool;
   // END_VAR
BEGIN
END_DATA_BLOCK

DATA_BLOCK "Tim 202"   // DB202
{ S7_Optimized_Access := 'TRUE' }
// stored: AutoNumber false, InstanceOfName IEC_TIMER, OfSystemLibElement IEC_TIMER, OfSystemLibVersion 1.0
"IEC_TIMER"
   // VAR
   //    PT : Time;
   //    ET { ExternalWritable := 'False'} : Time;
   //    IN : Bool;
   //    Q { ExternalWritable := 'False'} : Bool;
   // END_VAR
BEGIN
END_DATA_BLOCK

DATA_BLOCK "Tim 203"   // DB203
{ S7_Optimized_Access := 'TRUE' }
// stored: AutoNumber false, InstanceOfName IEC_TIMER, OfSystemLibElement IEC_TIMER, OfSystemLibVersion 1.0
"IEC_TIMER"
   // VAR
   //    PT : Time;
   //    ET { ExternalWritable := 'False'} : Time;
   //    IN : Bool;
   //    Q { ExternalWritable := 'False'} : Bool;
   // END_VAR
BEGIN
END_DATA_BLOCK

DATA_BLOCK "Tim 204"   // DB204
{ S7_Optimized_Access := 'TRUE' }
// stored: AutoNumber false, InstanceOfName IEC_TIMER, OfSystemLibElement IEC_TIMER, OfSystemLibVersion 1.0
"IEC_TIMER"
   // VAR
   //    PT : Time;
   //    ET { ExternalWritable := 'False'} : Time;
   //    IN : Bool;
   //    Q { ExternalWritable := 'False'} : Bool;
   // END_VAR
BEGIN
END_DATA_BLOCK

DATA_BLOCK "Tim 210"   // DB210
{ S7_Optimized_Access := 'TRUE' }
// stored: AutoNumber false, InstanceOfName IEC_TIMER, OfSystemLibElement IEC_TIMER, OfSystemLibVersion 1.0
"IEC_TIMER"
   // VAR
   //    PT : Time;
   //    ET { ExternalWritable := 'False'} : Time;
   //    IN : Bool;
   //    Q { ExternalWritable := 'False'} : Bool;
   // END_VAR
BEGIN
END_DATA_BLOCK

DATA_BLOCK "Tim 211"   // DB211
{ S7_Optimized_Access := 'TRUE' }
// stored: AutoNumber false, InstanceOfName IEC_TIMER, OfSystemLibElement IEC_TIMER, OfSystemLibVersion 1.0
"IEC_TIMER"
   // VAR
   //    PT : Time;
   //    ET { ExternalWritable := 'False'} : Time;
   //    IN : Bool;
   //    Q { ExternalWritable := 'False'} : Bool;
   // END_VAR
BEGIN
END_DATA_BLOCK

DATA_BLOCK "Tim 212"   // DB212
{ S7_Optimized_Access := 'TRUE' }
// stored: AutoNumber false, InstanceOfName IEC_TIMER, OfSystemLibElement IEC_TIMER, OfSystemLibVersion 1.0
"IEC_TIMER"
   // VAR
   //    PT : Time;
   //    ET { ExternalWritable := 'False'} : Time;
   //    IN : Bool;
   //    Q { ExternalWritable := 'False'} : Bool;
   // END_VAR
BEGIN
END_DATA_BLOCK
